LIN {X 0,Y 185.582,Z 221.367,A -85,B 0,C 180,E1 -22200.574,E2 -22200.574} C_VEL
LIN {X 0,Y 185.587,Z 221.368,A -85,B 0,C 180,E1 -22205.381,E2 -22205.381} C_VEL
LIN {X 0,Y 185.674,Z 221.358,A -85,B 0,C 180,E1 -22211.131,E2 -22211.131} C_VEL
LIN {X 0,Y 185.764,Z 221.345,A -85,B 0,C 180,E1 -22216.878,E2 -22216.878} C_VEL
LIN {X 0,Y 186.023,Z 221.31,A -85,B 0,C 180,E1 -22221.307,E2 -22221.307} C_VEL
LIN {X 0,Y 186.206,Z 221.287,A -85,B 0,C 180,E1 -22227.835,E2 -22227.835} C_VEL
LIN {X 0,Y 186.405,Z 221.26,A -85,B 0,C 180,E1 -22229.998,E2 -22229.998} C_VEL
LIN {X 0,Y 185.923,Z 221.325,A -85,B 0,C 180,E1 -22234.334,E2 -22234.334} C_VEL
LIN {X 0,Y 186.006,Z 221.311,A -85,B 0,C 180,E1 -22238.691,E2 -22238.691} C_VEL
LIN {X 0,Y 185.761,Z 221.346,A -85,B 0,C 180,E1 -22243.119,E2 -22243.119} C_VEL
LIN {X 0,Y 185.671,Z 221.357,A -85,B 0,C 180,E1 -22248.866,E2 -22248.866} C_VEL
LIN {X 0,Y 185.596,Z 221.363,A -85,B 0,C 180,E1 -22254.661,E2 -22254.661} C_VEL
LIN {X 0,Y 185.574,Z 221.368,A -85,B 0,C 180,E1 -22259.492,E2 -22259.492} C_VEL
LIN {X 0,Y 185.515,Z 221.375,A -85,B 0,C 180,E1 -22264.626,E2 -22264.626} C_VEL
LIN {X 0,Y 185.562,Z 221.369,A -85,B 0,C 180,E1 -22267.313,E2 -22267.313} C_VEL
LIN {X 0,Y 185.556,Z 221.367,A -85,B 0,C 180,E1 -22270.757,E2 -22270.757} C_VEL
LIN {X 0,Y 185.555,Z 221.371,A -85,B 0,C 180,E1 -22276.022,E2 -22276.022} C_VEL
LIN {X 0,Y 185.527,Z 221.371,A -85,B 0,C 180,E1 -22279.912,E2 -22279.912} C_VEL
LIN {X 0,Y 185.537,Z 221.373,A -85,B 0,C 180,E1 -22282.696,E2 -22282.696} C_VEL
LIN {X 0,Y 185.539,Z 221.371,A -85,B 0,C 180,E1 -22287.975,E2 -22287.975} C_VEL
LIN {X 0,Y 185.575,Z 221.368,A -85,B 0,C 180,E1 -22290.576,E2 -22290.576} C_VEL
LIN {X 0,Y 185.581,Z 221.366,A -85,B 0,C 180,E1 -22295.383,E2 -22295.383} C_VEL
LIN {X 0,Y 185.668,Z 221.356,A -85,B 0,C 180,E1 -22301.133,E2 -22301.133} C_VEL
LIN {X 0,Y 185.688,Z 221.35,A -85,B 0,C 180,E1 -22304.638,E2 -22304.638} C_VEL
LIN {X 0,Y 185.882,Z 221.33,A -85,B 0,C 180,E1 -22309.418,E2 -22309.418} C_VEL
LIN {X 0,Y 185.941,Z 221.32,A -85,B 0,C 180,E1 -22313.49,E2 -22313.49} C_VEL
LIN {X 0,Y 186.2,Z 221.292,A -85,B 0,C 180,E1 -22317.838,E2 -22317.838} C_VEL
LIN {X 0,Y 186.401,Z 221.264,A -85,B 0,C 180,E1 -22320.001,E2 -22320.001} C_VEL
LIN {X 0,Y 185.919,Z 221.324,A -85,B 0,C 180,E1 -22324.337,E2 -22324.337} C_VEL
LIN {X 0,Y 186.009,Z 221.312,A -85,B 0,C 180,E1 -22328.694,E2 -22328.694} C_VEL
LIN {X 0,Y 185.729,Z 221.348,A -85,B 0,C 180,E1 -22333.124,E2 -22333.124} C_VEL
LIN {X 0,Y 185.686,Z 221.352,A -85,B 0,C 180,E1 -22337.626,E2 -22337.626} C_VEL
LIN {X 0,Y 185.593,Z 221.365,A -85,B 0,C 180,E1 -22342.253,E2 -22342.253} C_VEL
LIN {X 0,Y 185.557,Z 221.368,A -85,B 0,C 180,E1 -22347.034,E2 -22347.034} C_VEL
LIN {X 0,Y 185.574,Z 221.37,A -85,B 0,C 180,E1 -22349.495,E2 -22349.495} C_VEL
LIN {X 0,Y 185.495,Z 221.379,A -85,B 0,C 180,E1 -22354.634,E2 -22354.634} C_VEL
LIN {X 0,Y 185.503,Z 221.379,A -85,B 0,C 180,E1 -22357.315,E2 -22357.315} C_VEL
LIN {X 0,Y 185.468,Z 221.383,A -85,B 0,C 180,E1 -22360.726,E2 -22360.726} C_VEL
LIN {X 0,Y 185.457,Z 221.384,A -85,B 0,C 180,E1 -22366.057,E2 -22366.057} C_VEL
LIN {X 0,Y 185.554,Z 221.623,A -85,B 0,C 180,E1 -22368.586,E2 -22368.586} C_VEL
LIN {X 0,Y 188.222,Z 233.304,A -85,B 0,C 180,E1 -22373.317,E2 -22373.317} C_VEL
LIN {X 0,Y 191.21,Z 247.009,A -85,B 0,C 180,E1 -22378.502,E2 -22378.502} C_VEL
LIN {X 0,Y 191.532,Z 248.614,A -85,B 0,C 180,E1 -22379.091,E2 -22379.091} C_VEL
LIN {X 0,Y 190.541,Z 254.381,A -85,B 0,C 180,E1 -22380.972,E2 -22380.972} C_VEL
LIN {X 0,Y 190.999,Z 275.587,A -85,B 0,C 180,E1 -22382.161,E2 -22382.161} C_VEL
LIN {X 0,Y 192.737,Z 304.014,A -85,B 0,C 180,E1 -22383.761,E2 -22383.761} C_VEL
LIN {X 0,Y 191.174,Z 343.448,A -85,B 0,C 180,E1 -22385.757,E2 -22385.757} C_VEL
LIN {X 0,Y 190.275,Z 349.218,A -85,B 0,C 180,E1 -22386.03,E2 -22386.03} C_VEL
LIN {X 0,Y 186.914,Z 358.417,A -85,B 0,C 180,E1 -22386.543,E2 -22386.543} C_VEL
LIN {X 0,Y 183.519,Z 367.45,A -85,B 0,C 180,E1 -22387.317,E2 -22387.317} C_VEL
LIN {X 0,Y 182.429,Z 372.966,A -85,B 0,C 180,E1 -22387.93,E2 -22387.93} C_VEL
LIN {X 0,Y 181.332,Z 384.689,A -85,B 0,C 180,E1 -22389.587,E2 -22389.587} C_VEL
LIN {X 0,Y 180.097,Z 396.698,A -85,B 0,C 180,E1 -22391.811,E2 -22391.811} C_VEL
LIN {X 0,Y 178.971,Z 407.243,A -85,B 0,C 180,E1 -22394.339,E2 -22394.339} C_VEL
LIN {X 0,Y 178.275,Z 415.873,A -85,B 0,C 180,E1 -22396.9,E2 -22396.9} C_VEL
LIN {X 0,Y 177.838,Z 423.688,A -85,B 0,C 180,E1 -22399.758,E2 -22399.758} C_VEL
LIN {X 0,Y 177.753,Z 431.165,A -85,B 0,C 180,E1 -22403.19,E2 -22403.19} C_VEL
LIN {X 0,Y 177.955,Z 436.97,A -85,B 0,C 180,E1 -22406.605,E2 -22406.605} C_VEL
LIN {X 0,Y 178.102,Z 441.236,A -85,B 0,C 180,E1 -22410.002,E2 -22410.002} C_VEL
LIN {X 0,Y 177.77,Z 443.242,A -85,B 0,C 180,E1 -22412.267,E2 -22412.267} C_VEL
LIN {X 0,Y 177.257,Z 444.744,A -85,B 0,C 180,E1 -22414.55,E2 -22414.55} C_VEL
LIN {X 0,Y 176.914,Z 445.823,A -85,B 0,C 180,E1 -22416.846,E2 -22416.846} C_VEL
LIN {X 0,Y 176.939,Z 446.736,A -85,B 0,C 180,E1 -22421.457,E2 -22421.457} C_VEL
LIN {X 0,Y 178.334,Z 446.179,A -85,B 0,C 180,E1 -22426.015,E2 -22426.015} C_VEL
LIN {X 0,Y 181.151,Z 444.075,A -85,B 0,C 180,E1 -22430.438,E2 -22430.438} C_VEL
LIN {X 0,Y 185.157,Z 440.45,A -85,B 0,C 180,E1 -22434.68,E2 -22434.68} C_VEL
LIN {X 0,Y 188.911,Z 436.629,A -85,B 0,C 180,E1 -22437.714,E2 -22437.714} C_VEL
LIN {X 0,Y 193.435,Z 431.743,A -85,B 0,C 180,E1 -22440.576,E2 -22440.576} C_VEL
LIN {X 0,Y 199.599,Z 424.531,A -85,B 0,C 180,E1 -22443.682,E2 -22443.682} C_VEL
LIN {X 0,Y 205.382,Z 416.886,A -85,B 0,C 180,E1 -22446.178,E2 -22446.178} C_VEL
LIN {X 0,Y 211.709,Z 407.374,A -85,B 0,C 180,E1 -22448.495,E2 -22448.495} C_VEL
LIN {X 0,Y 217.437,Z 397.694,A -85,B 0,C 180,E1 -22450.275,E2 -22450.275} C_VEL
LIN {X 0,Y 223.572,Z 385.631,A -85,B 0,C 180,E1 -22451.914,E2 -22451.914} C_VEL
LIN {X 0,Y 227.994,Z 375.107,A -85,B 0,C 180,E1 -22453.002,E2 -22453.002} C_VEL
LIN {X 0,Y 232.578,Z 361.508,A -85,B 0,C 180,E1 -22454.029,E2 -22454.029} C_VEL
LIN {X 0,Y 235.99,Z 347.508,A -85,B 0,C 180,E1 -22454.767,E2 -22454.767} C_VEL
LIN {X 0,Y 240.798,Z 317.9,A -85,B 0,C 180,E1 -22456.017,E2 -22456.017} C_VEL
LIN {X 0,Y 241.066,Z 314.821,A -85,B 0,C 180,E1 -22456.308,E2 -22456.308} C_VEL
LIN {X 0,Y 239.637,Z 310.317,A -85,B 0,C 180,E1 -22458.172,E2 -22458.172} C_VEL
LIN {X 0,Y 238.378,Z 306.264,A -85,B 0,C 180,E1 -22460.344,E2 -22460.344} C_VEL
LIN {X 0,Y 237.037,Z 302.381,A -85,B 0,C 180,E1 -22463.766,E2 -22463.766} C_VEL
LIN {X 0,Y 236.768,Z 301.25,A -85,B 0,C 180,E1 -22465.668,E2 -22465.668} C_VEL
LIN {X 0,Y 236.704,Z 300.974,A -85,B 0,C 180,E1 -22467.693,E2 -22467.693} C_VEL
LIN {X 0,Y 237.19,Z 301.52,A -85,B 0,C 180,E1 -22470.349,E2 -22470.349} C_VEL
LIN {X 0,Y 238.419,Z 303.667,A -85,B 0,C 180,E1 -22473.28,E2 -22473.28} C_VEL
LIN {X 0,Y 240.206,Z 307.592,A -85,B 0,C 180,E1 -22476.073,E2 -22476.073} C_VEL
LIN {X 0,Y 241.314,Z 310.279,A -85,B 0,C 180,E1 -22477.425,E2 -22477.425} C_VEL
LIN {X 0,Y 236.461,Z 338.426,A -85,B 0,C 180,E1 -22478.792,E2 -22478.792} C_VEL
LIN {X 0,Y 233.294,Z 351.201,A -85,B 0,C 180,E1 -22479.73,E2 -22479.73} C_VEL
LIN {X 0,Y 229.171,Z 363.637,A -85,B 0,C 180,E1 -22480.983,E2 -22480.983} C_VEL
LIN {X 0,Y 224.538,Z 374.681,A -85,B 0,C 180,E1 -22482.466,E2 -22482.466} C_VEL
LIN {X 0,Y 219.655,Z 384.181,A -85,B 0,C 180,E1 -22484.128,E2 -22484.128} C_VEL
LIN {X 0,Y 214.005,Z 393.392,A -85,B 0,C 180,E1 -22486.225,E2 -22486.225} C_VEL
LIN {X 0,Y 208.873,Z 400.55,A -85,B 0,C 180,E1 -22488.352,E2 -22488.352} C_VEL
LIN {X 0,Y 203.977,Z 406.361,A -85,B 0,C 180,E1 -22490.58,E2 -22490.58} C_VEL
LIN {X 0,Y 199.59,Z 410.86,A -85,B 0,C 180,E1 -22492.879,E2 -22492.879} C_VEL
LIN {X 0,Y 194.612,Z 415.134,A -85,B 0,C 180,E1 -22495.857,E2 -22495.857} C_VEL
LIN {X 0,Y 189.772,Z 418.269,A -85,B 0,C 180,E1 -22499.324,E2 -22499.324} C_VEL
LIN {X 0,Y 186.483,Z 419.638,A -85,B 0,C 180,E1 -22502.159,E2 -22502.159} C_VEL
LIN {X 0,Y 183.501,Z 420.12,A -85,B 0,C 180,E1 -22505.252,E2 -22505.252} C_VEL
LIN {X 0,Y 180.779,Z 419.378,A -85,B 0,C 180,E1 -22508.945,E2 -22508.945} C_VEL
LIN {X 0,Y 179.319,Z 418.115,A -85,B 0,C 180,E1 -22511.525,E2 -22511.525} C_VEL
LIN {X 0,Y 177.929,Z 415.513,A -85,B 0,C 180,E1 -22514.876,E2 -22514.876} C_VEL
LIN {X 0,Y 177.063,Z 411.424,A -85,B 0,C 180,E1 -22518.513,E2 -22518.513} C_VEL
LIN {X 0,Y 176.816,Z 405.855,A -85,B 0,C 180,E1 -22522.184,E2 -22522.184} C_VEL
LIN {X 0,Y 177.175,Z 398.545,A -85,B 0,C 180,E1 -22525.869,E2 -22525.869} C_VEL
LIN {X 0,Y 177.738,Z 390.602,A -85,B 0,C 180,E1 -22528.993,E2 -22528.993} C_VEL
LIN {X 0,Y 178.494,Z 381.753,A -85,B 0,C 180,E1 -22531.776,E2 -22531.776} C_VEL
LIN {X 0,Y 179.446,Z 371.889,A -85,B 0,C 180,E1 -22534.26,E2 -22534.26} C_VEL
LIN {X 0,Y 180.458,Z 361.055,A -85,B 0,C 180,E1 -22536.434,E2 -22536.434} C_VEL
LIN {X 0,Y 181.491,Z 349.211,A -85,B 0,C 180,E1 -22538.284,E2 -22538.284} C_VEL
LIN {X 0,Y 182.352,Z 337.137,A -85,B 0,C 180,E1 -22539.692,E2 -22539.692} C_VEL
LIN {X 0,Y 182.996,Z 323.953,A -85,B 0,C 180,E1 -22540.758,E2 -22540.758} C_VEL
LIN {X 0,Y 185.457,Z 265.599,A -85,B 0,C 180,E1 -22544.188,E2 -22544.188} C_VEL
LIN {X 0,Y 182.652,Z 241.648,A -85,B 0,C 180,E1 -22545.793,E2 -22545.793} C_VEL
LIN {X 0,Y 181.654,Z 237.511,A -85,B 0,C 180,E1 -22546.212,E2 -22546.212} C_VEL
LIN {X 0,Y 179.188,Z 225.225,A -85,B 0,C 180,E1 -22551.666,E2 -22551.666} C_VEL
LIN {X 0,Y 178.573,Z 222.387,A -85,B 0,C 180,E1 -22553.103,E2 -22553.103} C_VEL
LIN {X 0,Y 178.489,Z 222.252,A -85,B 0,C 180,E1 -22556.546,E2 -22556.546} C_VEL
LIN {X 0,Y 178.523,Z 222.248,A -85,B 0,C 180,E1 -22560.005,E2 -22560.005} C_VEL
LIN {X 0,Y 178.534,Z 222.244,A -85,B 0,C 180,E1 -22564.874,E2 -22564.874} C_VEL
LIN {X 0,Y 178.622,Z 222.235,A -85,B 0,C 180,E1 -22570.782,E2 -22570.782} C_VEL
LIN {X 0,Y 178.68,Z 222.226,A -85,B 0,C 180,E1 -22576.348,E2 -22576.348} C_VEL
LIN {X 0,Y 178.973,Z 222.188,A -85,B 0,C 180,E1 -22580.961,E2 -22580.961} C_VEL
LIN {X 0,Y 179.152,Z 222.166,A -85,B 0,C 180,E1 -22587.75,E2 -22587.75} C_VEL
LIN {X 0,Y 179.368,Z 222.137,A -85,B 0,C 180,E1 -22589.998,E2 -22589.998} C_VEL
LIN {X 0,Y 178.871,Z 222.204,A -85,B 0,C 180,E1 -22594.505,E2 -22594.505} C_VEL
LIN {X 0,Y 178.956,Z 222.191,A -85,B 0,C 180,E1 -22599.036,E2 -22599.036} C_VEL
LIN {X 0,Y 178.678,Z 222.226,A -85,B 0,C 180,E1 -22603.649,E2 -22603.649} C_VEL
LIN {X 0,Y 178.619,Z 222.235,A -85,B 0,C 180,E1 -22609.215,E2 -22609.215} C_VEL
LIN {X 0,Y 178.53,Z 222.243,A -85,B 0,C 180,E1 -22615.123,E2 -22615.123} C_VEL
LIN {X 0,Y 178.474,Z 222.252,A -85,B 0,C 180,E1 -22620.789,E2 -22620.789} C_VEL
LIN {X 0,Y 178.479,Z 222.248,A -85,B 0,C 180,E1 -22624.219,E2 -22624.219} C_VEL
LIN {X 0,Y 178.467,Z 222.252,A -85,B 0,C 180,E1 -22629.053,E2 -22629.053} C_VEL
LIN {X 0,Y 178.494,Z 222.246,A -85,B 0,C 180,E1 -22632.015,E2 -22632.015} C_VEL
LIN {X 0,Y 178.51,Z 222.248,A -85,B 0,C 180,E1 -22635.124,E2 -22635.124} C_VEL
LIN {X 0,Y 178.478,Z 222.251,A -85,B 0,C 180,E1 -22638.429,E2 -22638.429} C_VEL
LIN {X 0,Y 178.444,Z 222.257,A -85,B 0,C 180,E1 -22643.789,E2 -22643.789} C_VEL
LIN {X 0,Y 178.485,Z 222.25,A -85,B 0,C 180,E1 -22646.548,E2 -22646.548} C_VEL
LIN {X 0,Y 178.516,Z 222.246,A -85,B 0,C 180,E1 -22650.006,E2 -22650.006} C_VEL
LIN {X 0,Y 178.528,Z 222.244,A -85,B 0,C 180,E1 -22654.876,E2 -22654.876} C_VEL
LIN {X 0,Y 178.617,Z 222.234,A -85,B 0,C 180,E1 -22660.784,E2 -22660.784} C_VEL
LIN {X 0,Y 178.651,Z 222.229,A -85,B 0,C 180,E1 -22666.348,E2 -22666.348} C_VEL
LIN {X 0,Y 178.905,Z 222.198,A -85,B 0,C 180,E1 -22670.961,E2 -22670.961} C_VEL
LIN {X 0,Y 179.146,Z 222.171,A -85,B 0,C 180,E1 -22677.753,E2 -22677.753} C_VEL
LIN {X 0,Y 179.364,Z 222.141,A -85,B 0,C 180,E1 -22680.001,E2 -22680.001} C_VEL
LIN {X 0,Y 178.868,Z 222.202,A -85,B 0,C 180,E1 -22684.508,E2 -22684.508} C_VEL
LIN {X 0,Y 178.958,Z 222.191,A -85,B 0,C 180,E1 -22689.039,E2 -22689.039} C_VEL
LIN {X 0,Y 178.656,Z 222.232,A -85,B 0,C 180,E1 -22693.653,E2 -22693.653} C_VEL
LIN {X 0,Y 178.619,Z 222.231,A -85,B 0,C 180,E1 -22699.218,E2 -22699.218} C_VEL
LIN {X 0,Y 178.531,Z 222.247,A -85,B 0,C 180,E1 -22705.126,E2 -22705.126} C_VEL
LIN {X 0,Y 178.474,Z 222.254,A -85,B 0,C 180,E1 -22710.793,E2 -22710.793} C_VEL
LIN {X 0,Y 178.481,Z 222.252,A -85,B 0,C 180,E1 -22714.221,E2 -22714.221} C_VEL
LIN {X 0,Y 178.392,Z 222.264,A -85,B 0,C 180,E1 -22719.077,E2 -22719.077} C_VEL
LIN {X 0,Y 178.395,Z 222.263,A -85,B 0,C 180,E1 -22722.047,E2 -22722.047} C_VEL
LIN {X 0,Y 178.391,Z 222.265,A -85,B 0,C 180,E1 -22725.166,E2 -22725.166} C_VEL
LIN {X 0,Y 178.502,Z 222.537,A -85,B 0,C 180,E1 -22728.094,E2 -22728.094} C_VEL
LIN {X 0,Y 181.016,Z 233.563,A -85,B 0,C 180,E1 -22732.742,E2 -22732.742} C_VEL
LIN {X 0,Y 184.108,Z 247.761,A -85,B 0,C 180,E1 -22738.342,E2 -22738.342} C_VEL
LIN {X 0,Y 184.459,Z 249.623,A -85,B 0,C 180,E1 -22739.048,E2 -22739.048} C_VEL
LIN {X 0,Y 183.628,Z 253.91,A -85,B 0,C 180,E1 -22740.496,E2 -22740.496} C_VEL
LIN {X 0,Y 183.824,Z 271.879,A -85,B 0,C 180,E1 -22741.565,E2 -22741.565} C_VEL
LIN {X 0,Y 185.717,Z 304.253,A -85,B 0,C 180,E1 -22743.45,E2 -22743.45} C_VEL
LIN {X 0,Y 183.695,Z 355.631,A -85,B 0,C 180,E1 -22746.271,E2 -22746.271} C_VEL
LIN {X 0,Y 182.99,Z 367.173,A -85,B 0,C 180,E1 -22747.282,E2 -22747.282} C_VEL
LIN {X 0,Y 182.429,Z 372.966,A -85,B 0,C 180,E1 -22747.93,E2 -22747.93} C_VEL
LIN {X 0,Y 181.253,Z 378.336,A -85,B 0,C 180,E1 -22748.614,E2 -22748.614} C_VEL
LIN {X 0,Y 177.603,Z 386.618,A -85,B 0,C 180,E1 -22749.908,E2 -22749.908} C_VEL
LIN {X 0,Y 173.919,Z 394.533,A -85,B 0,C 180,E1 -22751.478,E2 -22751.478} C_VEL
LIN {X 0,Y 172.705,Z 399.312,A -85,B 0,C 180,E1 -22752.57,E2 -22752.57} C_VEL
LIN {X 0,Y 171.627,Z 409.102,A -85,B 0,C 180,E1 -22755.173,E2 -22755.173} C_VEL
LIN {X 0,Y 171.042,Z 418.092,A -85,B 0,C 180,E1 -22758.146,E2 -22758.146} C_VEL
LIN {X 0,Y 170.693,Z 425.475,A -85,B 0,C 180,E1 -22761.182,E2 -22761.182} C_VEL
LIN {X 0,Y 170.828,Z 432.261,A -85,B 0,C 180,E1 -22764.69,E2 -22764.69} C_VEL
LIN {X 0,Y 171.081,Z 436.784,A -85,B 0,C 180,E1 -22767.647,E2 -22767.647} C_VEL
LIN {X 0,Y 171.163,Z 439.627,A -85,B 0,C 180,E1 -22770.002,E2 -22770.002} C_VEL
LIN {X 0,Y 170.795,Z 441.824,A -85,B 0,C 180,E1 -22772.36,E2 -22772.36} C_VEL
LIN {X 0,Y 169.927,Z 444.564,A -85,B 0,C 180,E1 -22776.959,E2 -22776.959} C_VEL
LIN {X 0,Y 169.771,Z 445.424,A -85,B 0,C 180,E1 -22779.533,E2 -22779.533} C_VEL
LIN {X 0,Y 170.562,Z 445.861,A -85,B 0,C 180,E1 -22784.315,E2 -22784.315} C_VEL
LIN {X 0,Y 172.832,Z 444.823,A -85,B 0,C 180,E1 -22788.986,E2 -22788.986} C_VEL
LIN {X 0,Y 174.502,Z 443.763,A -85,B 0,C 180,E1 -22791.254,E2 -22791.254} C_VEL
LIN {X 0,Y 178.698,Z 440.432,A -85,B 0,C 180,E1 -22795.635,E2 -22795.635} C_VEL
LIN {X 0,Y 182.654,Z 436.866,A -85,B 0,C 180,E1 -22798.75,E2 -22798.75} C_VEL
LIN {X 0,Y 187.39,Z 432.327,A -85,B 0,C 180,E1 -22801.674,E2 -22801.674} C_VEL
LIN {X 0,Y 193.804,Z 425.594,A -85,B 0,C 180,E1 -22804.832,E2 -22804.832} C_VEL
LIN {X 0,Y 199.795,Z 418.312,A -85,B 0,C 180,E1 -22807.359,E2 -22807.359} C_VEL
LIN {X 0,Y 206.341,Z 409.483,A -85,B 0,C 180,E1 -22809.691,E2 -22809.691} C_VEL
LIN {X 0,Y 212.824,Z 399.443,A -85,B 0,C 180,E1 -22811.651,E2 -22811.651} C_VEL
LIN {X 0,Y 219.127,Z 388.06,A -85,B 0,C 180,E1 -22813.28,E2 -22813.28} C_VEL
LIN {X 0,Y 225.032,Z 375.094,A -85,B 0,C 180,E1 -22814.645,E2 -22814.645} C_VEL
LIN {X 0,Y 229.762,Z 361.936,A -85,B 0,C 180,E1 -22815.644,E2 -22815.644} C_VEL
LIN {X 0,Y 233.3,Z 348.771,A -85,B 0,C 180,E1 -22816.349,E2 -22816.349} C_VEL
LIN {X 0,Y 238.354,Z 319.482,A -85,B 0,C 180,E1 -22817.571,E2 -22817.571} C_VEL
LIN {X 0,Y 237.48,Z 316.125,A -85,B 0,C 180,E1 -22819.03,E2 -22819.03} C_VEL
LIN {X 0,Y 236.531,Z 312.836,A -85,B 0,C 180,E1 -22820.823,E2 -22820.823} C_VEL
LIN {X 0,Y 235.44,Z 309.191,A -85,B 0,C 180,E1 -22824.071,E2 -22824.071} C_VEL
LIN {X 0,Y 235.228,Z 308.105,A -85,B 0,C 180,E1 -22826,E2 -22826} C_VEL
LIN {X 0,Y 235.265,Z 307.946,A -85,B 0,C 180,E1 -22828.29,E2 -22828.29} C_VEL
LIN {X 0,Y 235.798,Z 308.729,A -85,B 0,C 180,E1 -22830.768,E2 -22830.768} C_VEL
LIN {X 0,Y 236.725,Z 310.562,A -85,B 0,C 180,E1 -22833.071,E2 -22833.071} C_VEL
LIN {X 0,Y 238.329,Z 314.413,A -85,B 0,C 180,E1 -22835.762,E2 -22835.762} C_VEL
LIN {X 0,Y 238.469,Z 314.81,A -85,B 0,C 180,E1 -22835.983,E2 -22835.983} C_VEL
LIN {X 0,Y 233.809,Z 340.377,A -85,B 0,C 180,E1 -22837.239,E2 -22837.239} C_VEL
LIN {X 0,Y 230.54,Z 352.77,A -85,B 0,C 180,E1 -22838.168,E2 -22838.168} C_VEL
LIN {X 0,Y 226.548,Z 364.138,A -85,B 0,C 180,E1 -22839.296,E2 -22839.296} C_VEL
LIN {X 0,Y 221.7,Z 375.004,A -85,B 0,C 180,E1 -22840.725,E2 -22840.725} C_VEL
LIN {X 0,Y 216.176,Z 385.248,A -85,B 0,C 180,E1 -22842.498,E2 -22842.498} C_VEL
LIN {X 0,Y 210.426,Z 394.163,A -85,B 0,C 180,E1 -22844.502,E2 -22844.502} C_VEL
LIN {X 0,Y 203.934,Z 402.509,A -85,B 0,C 180,E1 -22847.055,E2 -22847.055} C_VEL
LIN {X 0,Y 197.772,Z 409.059,A -85,B 0,C 180,E1 -22849.764,E2 -22849.764} C_VEL
LIN {X 0,Y 192.551,Z 413.748,A -85,B 0,C 180,E1 -22852.502,E2 -22852.502} C_VEL
LIN {X 0,Y 187.239,Z 417.47,A -85,B 0,C 180,E1 -22855.694,E2 -22855.694} C_VEL
LIN {X 0,Y 182.762,Z 419.768,A -85,B 0,C 180,E1 -22858.94,E2 -22858.94} C_VEL
LIN {X 0,Y 179.014,Z 420.831,A -85,B 0,C 180,E1 -22862.249,E2 -22862.249} C_VEL
LIN {X 0,Y 176.384,Z 420.838,A -85,B 0,C 180,E1 -22865.037,E2 -22865.037} C_VEL
LIN {X 0,Y 174.945,Z 420.446,A -85,B 0,C 180,E1 -22866.921,E2 -22866.921} C_VEL
LIN {X 0,Y 173.334,Z 419.463,A -85,B 0,C 180,E1 -22869.333,E2 -22869.333} C_VEL
LIN {X 0,Y 171.474,Z 416.992,A -85,B 0,C 180,E1 -22873.026,E2 -22873.026} C_VEL
LIN {X 0,Y 170.263,Z 413.258,A -85,B 0,C 180,E1 -22876.793,E2 -22876.793} C_VEL
LIN {X 0,Y 169.78,Z 408.067,A -85,B 0,C 180,E1 -22880.6,E2 -22880.6} C_VEL
LIN {X 0,Y 169.845,Z 402.477,A -85,B 0,C 180,E1 -22883.792,E2 -22883.792} C_VEL
LIN {X 0,Y 170.308,Z 395.497,A -85,B 0,C 180,E1 -22886.995,E2 -22886.995} C_VEL
LIN {X 0,Y 170.985,Z 386.404,A -85,B 0,C 180,E1 -22890.324,E2 -22890.324} C_VEL
LIN {X 0,Y 172.022,Z 375.426,A -85,B 0,C 180,E1 -22893.472,E2 -22893.472} C_VEL
LIN {X 0,Y 173.162,Z 363.57,A -85,B 0,C 180,E1 -22896.1,E2 -22896.1} C_VEL
LIN {X 0,Y 174.224,Z 351.436,A -85,B 0,C 180,E1 -22898.146,E2 -22898.146} C_VEL
LIN {X 0,Y 175.175,Z 338.681,A -85,B 0,C 180,E1 -22899.746,E2 -22899.746} C_VEL
LIN {X 0,Y 175.85,Z 326.101,A -85,B 0,C 180,E1 -22900.854,E2 -22900.854} C_VEL
LIN {X 0,Y 178.443,Z 266.016,A -85,B 0,C 180,E1 -22904.55,E2 -22904.55} C_VEL
LIN {X 0,Y 175.792,Z 243.119,A -85,B 0,C 180,E1 -22906.165,E2 -22906.165} C_VEL
LIN {X 0,Y 174.512,Z 237.87,A -85,B 0,C 180,E1 -22906.67,E2 -22906.67} C_VEL
LIN {X 0,Y 172.038,Z 225.846,A -85,B 0,C 180,E1 -22912.208,E2 -22912.208} C_VEL
LIN {X 0,Y 171.539,Z 223.201,A -85,B 0,C 180,E1 -22913.643,E2 -22913.643} C_VEL
LIN {X 0,Y 171.458,Z 223.129,A -85,B 0,C 180,E1 -22919.402,E2 -22919.402} C_VEL
LIN {X 0,Y 171.469,Z 223.124,A -85,B 0,C 180,E1 -22924.382,E2 -22924.382} C_VEL
LIN {X 0,Y 171.578,Z 223.112,A -85,B 0,C 180,E1 -22930.87,E2 -22930.87} C_VEL
LIN {X 0,Y 171.593,Z 223.11,A -85,B 0,C 180,E1 -22935.773,E2 -22935.773} C_VEL
LIN {X 0,Y 171.906,Z 223.068,A -85,B 0,C 180,E1 -22940.587,E2 -22940.587} C_VEL
LIN {X 0,Y 171.823,Z 223.083,A -85,B 0,C 180,E1 -22945.306,E2 -22945.306} C_VEL
LIN {X 0,Y 172.331,Z 223.013,A -85,B 0,C 180,E1 -22949.998,E2 -22949.998} C_VEL
LIN {X 0,Y 171.82,Z 223.083,A -85,B 0,C 180,E1 -22954.691,E2 -22954.691} C_VEL
LIN {X 0,Y 171.885,Z 223.072,A -85,B 0,C 180,E1 -22959.411,E2 -22959.411} C_VEL
LIN {X 0,Y 171.591,Z 223.109,A -85,B 0,C 180,E1 -22964.224,E2 -22964.224} C_VEL
LIN {X 0,Y 171.54,Z 223.116,A -85,B 0,C 180,E1 -22969.561,E2 -22969.561} C_VEL
LIN {X 0,Y 171.464,Z 223.122,A -85,B 0,C 180,E1 -22975.615,E2 -22975.615} C_VEL
LIN {X 0,Y 171.437,Z 223.13,A -85,B 0,C 180,E1 -22980.586,E2 -22980.586} C_VEL
LIN {X 0,Y 171.399,Z 223.133,A -85,B 0,C 180,E1 -22985.031,E2 -22985.031} C_VEL
LIN {X 0,Y 171.421,Z 223.131,A -85,B 0,C 180,E1 -22988.836,E2 -22988.836} C_VEL
LIN {X 0,Y 171.436,Z 223.129,A -85,B 0,C 180,E1 -22994.177,E2 -22994.177} C_VEL
LIN {X 0,Y 171.395,Z 223.131,A -85,B 0,C 180,E1 -22999,E2 -22999} C_VEL
LIN {X 0,Y 171.415,Z 223.131,A -85,B 0,C 180,E1 -23002.05,E2 -23002.05} C_VEL
LIN {X 0,Y 171.405,Z 223.133,A -85,B 0,C 180,E1 -23005.086,E2 -23005.086} C_VEL
LIN {X 0,Y 171.443,Z 223.128,A -85,B 0,C 180,E1 -23010.535,E2 -23010.535} C_VEL
LIN {X 0,Y 171.451,Z 223.126,A -85,B 0,C 180,E1 -23015.802,E2 -23015.802} C_VEL
LIN {X 0,Y 171.573,Z 223.112,A -85,B 0,C 180,E1 -23020.872,E2 -23020.872} C_VEL
LIN {X 0,Y 171.569,Z 223.109,A -85,B 0,C 180,E1 -23025.773,E2 -23025.773} C_VEL
LIN {X 0,Y 171.842,Z 223.078,A -85,B 0,C 180,E1 -23030.586,E2 -23030.586} C_VEL
LIN {X 0,Y 171.809,Z 223.08,A -85,B 0,C 180,E1 -23035.308,E2 -23035.308} C_VEL
LIN {X 0,Y 172.327,Z 223.017,A -85,B 0,C 180,E1 -23040.001,E2 -23040.001} C_VEL
LIN {X 0,Y 171.817,Z 223.081,A -85,B 0,C 180,E1 -23044.694,E2 -23044.694} C_VEL
LIN {X 0,Y 171.886,Z 223.071,A -85,B 0,C 180,E1 -23049.414,E2 -23049.414} C_VEL
LIN {X 0,Y 171.573,Z 223.112,A -85,B 0,C 180,E1 -23054.229,E2 -23054.229} C_VEL
LIN {X 0,Y 171.54,Z 223.114,A -85,B 0,C 180,E1 -23059.564,E2 -23059.564} C_VEL
LIN {X 0,Y 171.465,Z 223.124,A -85,B 0,C 180,E1 -23065.618,E2 -23065.618} C_VEL
LIN {X 0,Y 171.436,Z 223.13,A -85,B 0,C 180,E1 -23070.587,E2 -23070.587} C_VEL
LIN {X 0,Y 171.39,Z 223.138,A -85,B 0,C 180,E1 -23075.037,E2 -23075.037} C_VEL
LIN {X 0,Y 171.355,Z 223.14,A -85,B 0,C 180,E1 -23078.809,E2 -23078.809} C_VEL
LIN {X 0,Y 171.318,Z 223.145,A -85,B 0,C 180,E1 -23084.22,E2 -23084.22} C_VEL
LIN {X 0,Y 171.43,Z 223.387,A -85,B 0,C 180,E1 -23087.557,E2 -23087.557} C_VEL
LIN {X 0,Y 173.923,Z 234.398,A -85,B 0,C 180,E1 -23092.392,E2 -23092.392} C_VEL
LIN {X 0,Y 176.673,Z 246.948,A -85,B 0,C 180,E1 -23097.546,E2 -23097.546} C_VEL
LIN {X 0,Y 177.32,Z 250.582,A -85,B 0,C 180,E1 -23098.988,E2 -23098.988} C_VEL
LIN {X 0,Y 176.665,Z 253.766,A -85,B 0,C 180,E1 -23100.076,E2 -23100.076} C_VEL
LIN {X 0,Y 176.965,Z 275.277,A -85,B 0,C 180,E1 -23101.375,E2 -23101.375} C_VEL
LIN {X 0,Y 178.66,Z 304.843,A -85,B 0,C 180,E1 -23103.185,E2 -23103.185} C_VEL
LIN {X 0,Y 176.634,Z 355.237,A -85,B 0,C 180,E1 -23106.081,E2 -23106.081} C_VEL
LIN {X 0,Y 175.853,Z 367.669,A -85,B 0,C 180,E1 -23107.234,E2 -23107.234} C_VEL
LIN {X 0,Y 174.764,Z 379.495,A -85,B 0,C 180,E1 -23108.783,E2 -23108.783} C_VEL
LIN {X 0,Y 173.565,Z 391.128,A -85,B 0,C 180,E1 -23110.794,E2 -23110.794} C_VEL
LIN {X 0,Y 172.705,Z 399.312,A -85,B 0,C 180,E1 -23112.57,E2 -23112.57} C_VEL
LIN {X 0,Y 171.497,Z 403.924,A -85,B 0,C 180,E1 -23113.744,E2 -23113.744} C_VEL
LIN {X 0,Y 167.932,Z 410.724,A -85,B 0,C 180,E1 -23115.871,E2 -23115.871} C_VEL
LIN {X 0,Y 164.649,Z 417.032,A -85,B 0,C 180,E1 -23118.28,E2 -23118.28} C_VEL
LIN {X 0,Y 163.89,Z 420.781,A -85,B 0,C 180,E1 -23119.851,E2 -23119.851} C_VEL
LIN {X 0,Y 163.813,Z 427.926,A -85,B 0,C 180,E1 -23123.226,E2 -23123.226} C_VEL
LIN {X 0,Y 163.994,Z 433.162,A -85,B 0,C 180,E1 -23126.316,E2 -23126.316} C_VEL
LIN {X 0,Y 164.224,Z 436.539,A -85,B 0,C 180,E1 -23128.776,E2 -23128.776} C_VEL
LIN {X 0,Y 164.07,Z 439.23,A -85,B 0,C 180,E1 -23131.229,E2 -23131.229} C_VEL
LIN {X 0,Y 163.265,Z 442.071,A -85,B 0,C 180,E1 -23134.941,E2 -23134.941} C_VEL
LIN {X 0,Y 162.898,Z 443.394,A -85,B 0,C 180,E1 -23137.438,E2 -23137.438} C_VEL
LIN {X 0,Y 163.031,Z 444.836,A -85,B 0,C 180,E1 -23142.449,E2 -23142.449} C_VEL
LIN {X 0,Y 164.701,Z 444.853,A -85,B 0,C 180,E1 -23147.381,E2 -23147.381} C_VEL
LIN {X 0,Y 167.872,Z 443.361,A -85,B 0,C 180,E1 -23152.136,E2 -23152.136} C_VEL
LIN {X 0,Y 172.304,Z 440.396,A -85,B 0,C 180,E1 -23156.66,E2 -23156.66} C_VEL
LIN {X 0,Y 176.472,Z 437.138,A -85,B 0,C 180,E1 -23159.857,E2 -23159.857} C_VEL
LIN {X 0,Y 181.421,Z 432.9,A -85,B 0,C 180,E1 -23162.845,E2 -23162.845} C_VEL
LIN {X 0,Y 188.073,Z 426.539,A -85,B 0,C 180,E1 -23166.056,E2 -23166.056} C_VEL
LIN {X 0,Y 195.386,Z 418.545,A -85,B 0,C 180,E1 -23169.012,E2 -23169.012} C_VEL
LIN {X 0,Y 202.217,Z 409.905,A -85,B 0,C 180,E1 -23171.327,E2 -23171.327} C_VEL
LIN {X 0,Y 208.325,Z 401.157,A -85,B 0,C 180,E1 -23173.091,E2 -23173.091} C_VEL
LIN {X 0,Y 214.867,Z 390.474,A -85,B 0,C 180,E1 -23174.688,E2 -23174.688} C_VEL
LIN {X 0,Y 220.892,Z 378.54,A -85,B 0,C 180,E1 -23176.043,E2 -23176.043} C_VEL
LIN {X 0,Y 225.779,Z 366.558,A -85,B 0,C 180,E1 -23177.014,E2 -23177.014} C_VEL
LIN {X 0,Y 229.494,Z 354.984,A -85,B 0,C 180,E1 -23177.726,E2 -23177.726} C_VEL
LIN {X 0,Y 232.917,Z 340.14,A -85,B 0,C 180,E1 -23178.4,E2 -23178.4} C_VEL
LIN {X 0,Y 235.831,Z 323.61,A -85,B 0,C 180,E1 -23179.051,E2 -23179.051} C_VEL
LIN {X 0,Y 234.755,Z 319.39,A -85,B 0,C 180,E1 -23181.322,E2 -23181.322} C_VEL
LIN {X 0,Y 233.865,Z 315.922,A -85,B 0,C 180,E1 -23184.463,E2 -23184.463} C_VEL
LIN {X 0,Y 233.706,Z 315.024,A -85,B 0,C 180,E1 -23186.107,E2 -23186.107} C_VEL
LIN {X 0,Y 233.9,Z 315.046,A -85,B 0,C 180,E1 -23189.282,E2 -23189.282} C_VEL
LIN {X 0,Y 234.601,Z 316.36,A -85,B 0,C 180,E1 -23191.709,E2 -23191.709} C_VEL
LIN {X 0,Y 235.172,Z 317.943,A -85,B 0,C 180,E1 -23193.21,E2 -23193.21} C_VEL
LIN {X 0,Y 235.917,Z 319.667,A -85,B 0,C 180,E1 -23194.519,E2 -23194.519} C_VEL
LIN {X 0,Y 231.768,Z 341.207,A -85,B 0,C 180,E1 -23195.583,E2 -23195.583} C_VEL
LIN {X 0,Y 228.525,Z 352.861,A -85,B 0,C 180,E1 -23196.433,E2 -23196.433} C_VEL
LIN {X 0,Y 223.945,Z 365.222,A -85,B 0,C 180,E1 -23197.633,E2 -23197.633} C_VEL
LIN {X 0,Y 218.891,Z 376.078,A -85,B 0,C 180,E1 -23199.032,E2 -23199.032} C_VEL
LIN {X 0,Y 213.175,Z 386.092,A -85,B 0,C 180,E1 -23200.75,E2 -23200.75} C_VEL
LIN {X 0,Y 206.786,Z 395.306,A -85,B 0,C 180,E1 -23202.824,E2 -23202.824} C_VEL
LIN {X 0,Y 200.216,Z 403.332,A -85,B 0,C 180,E1 -23205.256,E2 -23205.256} C_VEL
LIN {X 0,Y 194.201,Z 409.37,A -85,B 0,C 180,E1 -23207.721,E2 -23207.721} C_VEL
LIN {X 0,Y 188.725,Z 413.993,A -85,B 0,C 180,E1 -23210.352,E2 -23210.352} C_VEL
LIN {X 0,Y 182.89,Z 417.964,A -85,B 0,C 180,E1 -23213.603,E2 -23213.603} C_VEL
LIN {X 0,Y 179.865,Z 419.563,A -85,B 0,C 180,E1 -23215.517,E2 -23215.517} C_VEL
LIN {X 0,Y 175.762,Z 421.116,A -85,B 0,C 180,E1 -23218.51,E2 -23218.51} C_VEL
LIN {X 0,Y 171.494,Z 421.763,A -85,B 0,C 180,E1 -23222.348,E2 -23222.348} C_VEL
LIN {X 0,Y 169.266,Z 421.437,A -85,B 0,C 180,E1 -23224.79,E2 -23224.79} C_VEL
LIN {X 0,Y 167.454,Z 420.637,A -85,B 0,C 180,E1 -23227.232,E2 -23227.232} C_VEL
LIN {X 0,Y 164.968,Z 418.05,A -85,B 0,C 180,E1 -23231.516,E2 -23231.516} C_VEL
LIN {X 0,Y 163.644,Z 414.938,A -85,B 0,C 180,E1 -23234.931,E2 -23234.931} C_VEL
LIN {X 0,Y 162.824,Z 409.74,A -85,B 0,C 180,E1 -23239.149,E2 -23239.149} C_VEL
LIN {X 0,Y 162.741,Z 402.728,A -85,B 0,C 180,E1 -23243.412,E2 -23243.412} C_VEL
LIN {X 0,Y 163.211,Z 395.336,A -85,B 0,C 180,E1 -23246.88,E2 -23246.88} C_VEL
LIN {X 0,Y 163.89,Z 386.307,A -85,B 0,C 180,E1 -23250.255,E2 -23250.255} C_VEL
LIN {X 0,Y 164.822,Z 376.188,A -85,B 0,C 180,E1 -23253.26,E2 -23253.26} C_VEL
LIN {X 0,Y 165.955,Z 364.47,A -85,B 0,C 180,E1 -23255.985,E2 -23255.985} C_VEL
LIN {X 0,Y 167.126,Z 351.664,A -85,B 0,C 180,E1 -23258.259,E2 -23258.259} C_VEL
LIN {X 0,Y 168.13,Z 338.345,A -85,B 0,C 180,E1 -23259.991,E2 -23259.991} C_VEL
LIN {X 0,Y 168.844,Z 325.1,A -85,B 0,C 180,E1 -23261.171,E2 -23261.171} C_VEL
LIN {X 0,Y 171.463,Z 266.646,A -85,B 0,C 180,E1 -23264.92,E2 -23264.92} C_VEL
LIN {X 0,Y 168.88,Z 244.508,A -85,B 0,C 180,E1 -23266.53,E2 -23266.53} C_VEL
LIN {X 0,Y 167.382,Z 238.271,A -85,B 0,C 180,E1 -23267.129,E2 -23267.129} C_VEL
LIN {X 0,Y 164.992,Z 226.774,A -85,B 0,C 180,E1 -23272.626,E2 -23272.626} C_VEL
LIN {X 0,Y 164.475,Z 224.096,A -85,B 0,C 180,E1 -23274.124,E2 -23274.124} C_VEL
LIN {X 0,Y 164.406,Z 224.007,A -85,B 0,C 180,E1 -23279.136,E2 -23279.136} C_VEL
LIN {X 0,Y 164.416,Z 224.002,A -85,B 0,C 180,E1 -23284.692,E2 -23284.692} C_VEL
LIN {X 0,Y 164.484,Z 223.996,A -85,B 0,C 180,E1 -23290.049,E2 -23290.049} C_VEL
LIN {X 0,Y 164.535,Z 223.988,A -85,B 0,C 180,E1 -23295.149,E2 -23295.149} C_VEL
LIN {X 0,Y 164.849,Z 223.946,A -85,B 0,C 180,E1 -23300.18,E2 -23300.18} C_VEL
LIN {X 0,Y 164.773,Z 223.961,A -85,B 0,C 180,E1 -23305.105,E2 -23305.105} C_VEL
LIN {X 0,Y 165.293,Z 223.89,A -85,B 0,C 180,E1 -23309.998,E2 -23309.998} C_VEL
LIN {X 0,Y 164.77,Z 223.962,A -85,B 0,C 180,E1 -23314.892,E2 -23314.892} C_VEL
LIN {X 0,Y 164.848,Z 223.945,A -85,B 0,C 180,E1 -23317.346,E2 -23317.346} C_VEL
LIN {X 0,Y 164.75,Z 223.964,A -85,B 0,C 180,E1 -23321.15,E2 -23321.15} C_VEL
LIN {X 0,Y 164.481,Z 223.993,A -85,B 0,C 180,E1 -23327.401,E2 -23327.401} C_VEL
LIN {X 0,Y 164.469,Z 223.997,A -85,B 0,C 180,E1 -23329.988,E2 -23329.988} C_VEL
LIN {X 0,Y 164.389,Z 224.004,A -85,B 0,C 180,E1 -23336.133,E2 -23336.133} C_VEL
LIN {X 0,Y 164.371,Z 224.007,A -85,B 0,C 180,E1 -23341.227,E2 -23341.227} C_VEL
LIN {X 0,Y 164.342,Z 224.014,A -85,B 0,C 180,E1 -23346.774,E2 -23346.774} C_VEL
LIN {X 0,Y 164.363,Z 224.009,A -85,B 0,C 180,E1 -23349.893,E2 -23349.893} C_VEL
LIN {X 0,Y 164.373,Z 224.007,A -85,B 0,C 180,E1 -23353.378,E2 -23353.378} C_VEL
LIN {X 0,Y 164.372,Z 224.009,A -85,B 0,C 180,E1 -23356.836,E2 -23356.836} C_VEL
LIN {X 0,Y 164.333,Z 224.011,A -85,B 0,C 180,E1 -23360.333,E2 -23360.333} C_VEL
LIN {X 0,Y 164.338,Z 224.015,A -85,B 0,C 180,E1 -23364.341,E2 -23364.341} C_VEL
LIN {X 0,Y 164.384,Z 224.003,A -85,B 0,C 180,E1 -23369.135,E2 -23369.135} C_VEL
LIN {X 0,Y 164.41,Z 224.003,A -85,B 0,C 180,E1 -23374.694,E2 -23374.694} C_VEL
LIN {X 0,Y 164.478,Z 223.998,A -85,B 0,C 180,E1 -23380.051,E2 -23380.051} C_VEL
LIN {X 0,Y 164.499,Z 223.989,A -85,B 0,C 180,E1 -23385.148,E2 -23385.148} C_VEL
LIN {X 0,Y 164.762,Z 223.961,A -85,B 0,C 180,E1 -23390.177,E2 -23390.177} C_VEL
LIN {X 0,Y 164.825,Z 223.949,A -85,B 0,C 180,E1 -23392.652,E2 -23392.652} C_VEL
LIN {X 0,Y 165.041,Z 223.927,A -85,B 0,C 180,E1 -23397.561,E2 -23397.561} C_VEL
LIN {X 0,Y 165.289,Z 223.894,A -85,B 0,C 180,E1 -23400.001,E2 -23400.001} C_VEL
LIN {X 0,Y 164.767,Z 223.959,A -85,B 0,C 180,E1 -23404.895,E2 -23404.895} C_VEL
LIN {X 0,Y 164.849,Z 223.951,A -85,B 0,C 180,E1 -23407.349,E2 -23407.349} C_VEL
LIN {X 0,Y 164.738,Z 223.959,A -85,B 0,C 180,E1 -23411.133,E2 -23411.133} C_VEL
LIN {X 0,Y 164.479,Z 223.994,A -85,B 0,C 180,E1 -23417.405,E2 -23417.405} C_VEL
LIN {X 0,Y 164.469,Z 223.995,A -85,B 0,C 180,E1 -23419.991,E2 -23419.991} C_VEL
LIN {X 0,Y 164.389,Z 224.004,A -85,B 0,C 180,E1 -23426.135,E2 -23426.135} C_VEL
LIN {X 0,Y 164.37,Z 224.01,A -85,B 0,C 180,E1 -23431.229,E2 -23431.229} C_VEL
LIN {X 0,Y 164.291,Z 224.019,A -85,B 0,C 180,E1 -23436.792,E2 -23436.792} C_VEL
LIN {X 0,Y 164.288,Z 224.02,A -85,B 0,C 180,E1 -23439.918,E2 -23439.918} C_VEL
LIN {X 0,Y 164.277,Z 224.023,A -85,B 0,C 180,E1 -23443.344,E2 -23443.344} C_VEL
LIN {X 0,Y 164.328,Z 224.239,A -85,B 0,C 180,E1 -23446.994,E2 -23446.994} C_VEL
LIN {X 0,Y 166.636,Z 234.161,A -85,B 0,C 180,E1 -23451.571,E2 -23451.571} C_VEL
LIN {X 0,Y 169.164,Z 245.79,A -85,B 0,C 180,E1 -23456.583,E2 -23456.583} C_VEL
LIN {X 0,Y 170.003,Z 249.655,A -85,B 0,C 180,E1 -23458.193,E2 -23458.193} C_VEL
LIN {X 0,Y 170.128,Z 251.436,A -85,B 0,C 180,E1 -23458.913,E2 -23458.913} C_VEL
LIN {X 0,Y 169.714,Z 253.47,A -85,B 0,C 180,E1 -23459.605,E2 -23459.605} C_VEL
LIN {X 0,Y 169.916,Z 274.41,A -85,B 0,C 180,E1 -23460.924,E2 -23460.924} C_VEL
LIN {X 0,Y 171.599,Z 305.412,A -85,B 0,C 180,E1 -23462.896,E2 -23462.896} C_VEL
LIN {X 0,Y 169.591,Z 354.558,A -85,B 0,C 180,E1 -23465.854,E2 -23465.854} C_VEL
LIN {X 0,Y 168.798,Z 367.26,A -85,B 0,C 180,E1 -23467.085,E2 -23467.085} C_VEL
LIN {X 0,Y 167.646,Z 379.627,A -85,B 0,C 180,E1 -23468.805,E2 -23468.805} C_VEL
LIN {X 0,Y 166.459,Z 391.043,A -85,B 0,C 180,E1 -23470.903,E2 -23470.903} C_VEL
LIN {X 0,Y 165.198,Z 402.437,A -85,B 0,C 180,E1 -23473.631,E2 -23473.631} C_VEL
LIN {X 0,Y 164.359,Z 411.64,A -85,B 0,C 180,E1 -23476.4,E2 -23476.4} C_VEL
LIN {X 0,Y 163.89,Z 420.781,A -85,B 0,C 180,E1 -23479.851,E2 -23479.851} C_VEL
LIN {X 0,Y 163.229,Z 424.335,A -85,B 0,C 180,E1 -23481.485,E2 -23481.485} C_VEL
LIN {X 0,Y 161.721,Z 427.409,A -85,B 0,C 180,E1 -23483.198,E2 -23483.198} C_VEL
LIN {X 0,Y 158.265,Z 432.551,A -85,B 0,C 180,E1 -23486.89,E2 -23486.89} C_VEL
LIN {X 0,Y 157.297,Z 435.688,A -85,B 0,C 180,E1 -23489.542,E2 -23489.542} C_VEL
LIN {X 0,Y 156.931,Z 438.719,A -85,B 0,C 180,E1 -23492.569,E2 -23492.569} C_VEL
LIN {X 0,Y 155.957,Z 441.921,A -85,B 0,C 180,E1 -23497.511,E2 -23497.511} C_VEL
LIN {X 0,Y 155.831,Z 443.12,A -85,B 0,C 180,E1 -23500.395,E2 -23500.395} C_VEL
LIN {X 0,Y 156.825,Z 444.116,A -85,B 0,C 180,E1 -23505.6,E2 -23505.6} C_VEL
LIN {X 0,Y 159.416,Z 443.679,A -85,B 0,C 180,E1 -23510.653,E2 -23510.653} C_VEL
LIN {X 0,Y 163.44,Z 441.802,A -85,B 0,C 180,E1 -23515.469,E2 -23515.469} C_VEL
LIN {X 0,Y 168.793,Z 438.404,A -85,B 0,C 180,E1 -23519.978,E2 -23519.978} C_VEL
LIN {X 0,Y 173.739,Z 434.79,A -85,B 0,C 180,E1 -23523.101,E2 -23523.101} C_VEL
LIN {X 0,Y 179.37,Z 430.216,A -85,B 0,C 180,E1 -23525.997,E2 -23525.997} C_VEL
LIN {X 0,Y 186.697,Z 423.431,A -85,B 0,C 180,E1 -23529.091,E2 -23529.091} C_VEL
LIN {X 0,Y 194.641,Z 414.806,A -85,B 0,C 180,E1 -23531.913,E2 -23531.913} C_VEL
LIN {X 0,Y 200.79,Z 407.285,A -85,B 0,C 180,E1 -23533.733,E2 -23533.733} C_VEL
LIN {X 0,Y 207.282,Z 398.176,A -85,B 0,C 180,E1 -23535.4,E2 -23535.4} C_VEL
LIN {X 0,Y 214.103,Z 386.953,A -85,B 0,C 180,E1 -23536.918,E2 -23536.918} C_VEL
LIN {X 0,Y 219.743,Z 375.844,A -85,B 0,C 180,E1 -23538.04,E2 -23538.04} C_VEL
LIN {X 0,Y 224.932,Z 363.191,A -85,B 0,C 180,E1 -23538.992,E2 -23538.992} C_VEL
LIN {X 0,Y 229.107,Z 349.736,A -85,B 0,C 180,E1 -23539.702,E2 -23539.702} C_VEL
LIN {X 0,Y 232.643,Z 332.43,A -85,B 0,C 180,E1 -23540.406,E2 -23540.406} C_VEL
LIN {X 0,Y 233.388,Z 328.135,A -85,B 0,C 180,E1 -23540.621,E2 -23540.621} C_VEL
LIN {X 0,Y 232.923,Z 325.653,A -85,B 0,C 180,E1 -23542.07,E2 -23542.07} C_VEL
LIN {X 0,Y 232.293,Z 322.637,A -85,B 0,C 180,E1 -23544.91,E2 -23544.91} C_VEL
LIN {X 0,Y 232.222,Z 322.027,A -85,B 0,C 180,E1 -23545.861,E2 -23545.861} C_VEL
LIN {X 0,Y 232.399,Z 322.043,A -85,B 0,C 180,E1 -23549.427,E2 -23549.427} C_VEL
LIN {X 0,Y 233.179,Z 323.693,A -85,B 0,C 180,E1 -23552.068,E2 -23552.068} C_VEL
LIN {X 0,Y 233.511,Z 324.893,A -85,B 0,C 180,E1 -23553.039,E2 -23553.039} C_VEL
LIN {X 0,Y 229.81,Z 342.859,A -85,B 0,C 180,E1 -23553.937,E2 -23553.937} C_VEL
LIN {X 0,Y 226.366,Z 354.498,A -85,B 0,C 180,E1 -23554.781,E2 -23554.781} C_VEL
LIN {X 0,Y 221.751,Z 366.334,A -85,B 0,C 180,E1 -23555.917,E2 -23555.917} C_VEL
LIN {X 0,Y 216.046,Z 377.769,A -85,B 0,C 180,E1 -23557.381,E2 -23557.381} C_VEL
LIN {X 0,Y 209.394,Z 388.569,A -85,B 0,C 180,E1 -23559.261,E2 -23559.261} C_VEL
LIN {X 0,Y 202.759,Z 397.415,A -85,B 0,C 180,E1 -23561.298,E2 -23561.298} C_VEL
LIN {X 0,Y 196.735,Z 404.194,A -85,B 0,C 180,E1 -23563.393,E2 -23563.393} C_VEL
LIN {X 0,Y 189.825,Z 410.684,A -85,B 0,C 180,E1 -23566.074,E2 -23566.074} C_VEL
LIN {X 0,Y 183.477,Z 415.601,A -85,B 0,C 180,E1 -23568.957,E2 -23568.957} C_VEL
LIN {X 0,Y 176.789,Z 419.53,A -85,B 0,C 180,E1 -23572.561,E2 -23572.561} C_VEL
LIN {X 0,Y 172.458,Z 421.368,A -85,B 0,C 180,E1 -23575.324,E2 -23575.324} C_VEL
LIN {X 0,Y 168.774,Z 422.334,A -85,B 0,C 180,E1 -23578.042,E2 -23578.042} C_VEL
LIN {X 0,Y 163.966,Z 422.425,A -85,B 0,C 180,E1 -23582.455,E2 -23582.455} C_VEL
LIN {X 0,Y 161.782,Z 421.729,A -85,B 0,C 180,E1 -23584.983,E2 -23584.983} C_VEL
LIN {X 0,Y 159.966,Z 420.555,A -85,B 0,C 180,E1 -23587.573,E2 -23587.573} C_VEL
LIN {X 0,Y 157.8,Z 417.794,A -85,B 0,C 180,E1 -23591.524,E2 -23591.524} C_VEL
LIN {X 0,Y 156.302,Z 413.699,A -85,B 0,C 180,E1 -23595.65,E2 -23595.65} C_VEL
LIN {X 0,Y 155.671,Z 408.202,A -85,B 0,C 180,E1 -23599.789,E2 -23599.789} C_VEL
LIN {X 0,Y 155.715,Z 401.003,A -85,B 0,C 180,E1 -23603.965,E2 -23603.965} C_VEL
LIN {X 0,Y 156.234,Z 393.404,A -85,B 0,C 180,E1 -23607.456,E2 -23607.456} C_VEL
LIN {X 0,Y 156.994,Z 383.962,A -85,B 0,C 180,E1 -23610.931,E2 -23610.931} C_VEL
LIN {X 0,Y 158.044,Z 372.697,A -85,B 0,C 180,E1 -23614.152,E2 -23614.152} C_VEL
LIN {X 0,Y 159.123,Z 361.733,A -85,B 0,C 180,E1 -23616.601,E2 -23616.601} C_VEL
LIN {X 0,Y 160.207,Z 349.677,A -85,B 0,C 180,E1 -23618.69,E2 -23618.69} C_VEL
LIN {X 0,Y 161.159,Z 336.801,A -85,B 0,C 180,E1 -23620.338,E2 -23620.338} C_VEL
LIN {X 0,Y 161.818,Z 323.93,A -85,B 0,C 180,E1 -23621.47,E2 -23621.47} C_VEL
LIN {X 0,Y 164.494,Z 267.338,A -85,B 0,C 180,E1 -23625.28,E2 -23625.28} C_VEL
LIN {X 0,Y 162.036,Z 245.966,A -85,B 0,C 180,E1 -23626.911,E2 -23626.911} C_VEL
LIN {X 0,Y 160.206,Z 238.603,A -85,B 0,C 180,E1 -23627.628,E2 -23627.628} C_VEL
LIN {X 0,Y 157.864,Z 227.296,A -85,B 0,C 180,E1 -23633.257,E2 -23633.257} C_VEL
LIN {X 0,Y 157.414,Z 225.07,A -85,B 0,C 180,E1 -23634.519,E2 -23634.519} C_VEL
LIN {X 0,Y 157.28,Z 224.893,A -85,B 0,C 180,E1 -23640.557,E2 -23640.557} C_VEL
LIN {X 0,Y 157.322,Z 224.889,A -85,B 0,C 180,E1 -23643.464,E2 -23643.464} C_VEL
LIN {X 0,Y 157.393,Z 224.88,A -85,B 0,C 180,E1 -23649.665,E2 -23649.665} C_VEL
LIN {X 0,Y 157.461,Z 224.867,A -85,B 0,C 180,E1 -23654.465,E2 -23654.465} C_VEL
LIN {X 0,Y 157.769,Z 224.829,A -85,B 0,C 180,E1 -23659.734,E2 -23659.734} C_VEL
LIN {X 0,Y 157.82,Z 224.822,A -85,B 0,C 180,E1 -23662.321,E2 -23662.321} C_VEL
LIN {X 0,Y 158.256,Z 224.766,A -85,B 0,C 180,E1 -23669.998,E2 -23669.998} C_VEL
LIN {X 0,Y 157.806,Z 224.822,A -85,B 0,C 180,E1 -23677.676,E2 -23677.676} C_VEL
LIN {X 0,Y 157.679,Z 224.844,A -85,B 0,C 180,E1 -23681.319,E2 -23681.319} C_VEL
LIN {X 0,Y 157.458,Z 224.866,A -85,B 0,C 180,E1 -23685.532,E2 -23685.532} C_VEL
LIN {X 0,Y 157.366,Z 224.883,A -85,B 0,C 180,E1 -23690.931,E2 -23690.931} C_VEL
LIN {X 0,Y 157.31,Z 224.888,A -85,B 0,C 180,E1 -23696.684,E2 -23696.684} C_VEL
LIN {X 0,Y 157.272,Z 224.891,A -85,B 0,C 180,E1 -23702.426,E2 -23702.426} C_VEL
LIN {X 0,Y 157.317,Z 224.889,A -85,B 0,C 180,E1 -23706.475,E2 -23706.475} C_VEL
LIN {X 0,Y 157.281,Z 224.888,A -85,B 0,C 180,E1 -23712.084,E2 -23712.084} C_VEL
LIN {X 0,Y 157.293,Z 224.891,A -85,B 0,C 180,E1 -23715.631,E2 -23715.631} C_VEL
LIN {X 0,Y 157.26,Z 224.892,A -85,B 0,C 180,E1 -23721.271,E2 -23721.271} C_VEL
LIN {X 0,Y 157.286,Z 224.893,A -85,B 0,C 180,E1 -23724.489,E2 -23724.489} C_VEL
LIN {X 0,Y 157.288,Z 224.888,A -85,B 0,C 180,E1 -23728.095,E2 -23728.095} C_VEL
LIN {X 0,Y 157.315,Z 224.888,A -85,B 0,C 180,E1 -23733.466,E2 -23733.466} C_VEL
LIN {X 0,Y 157.387,Z 224.879,A -85,B 0,C 180,E1 -23739.668,E2 -23739.668} C_VEL
LIN {X 0,Y 157.436,Z 224.869,A -85,B 0,C 180,E1 -23744.465,E2 -23744.465} C_VEL
LIN {X 0,Y 157.683,Z 224.844,A -85,B 0,C 180,E1 -23749.732,E2 -23749.732} C_VEL
LIN {X 0,Y 157.761,Z 224.829,A -85,B 0,C 180,E1 -23752.321,E2 -23752.321} C_VEL
LIN {X 0,Y 158.251,Z 224.77,A -85,B 0,C 180,E1 -23760.001,E2 -23760.001} C_VEL
LIN {X 0,Y 157.805,Z 224.828,A -85,B 0,C 180,E1 -23767.679,E2 -23767.679} C_VEL
LIN {X 0,Y 157.668,Z 224.84,A -85,B 0,C 180,E1 -23771.304,E2 -23771.304} C_VEL
LIN {X 0,Y 157.45,Z 224.873,A -85,B 0,C 180,E1 -23775.536,E2 -23775.536} C_VEL
LIN {X 0,Y 157.366,Z 224.88,A -85,B 0,C 180,E1 -23780.935,E2 -23780.935} C_VEL
LIN {X 0,Y 157.31,Z 224.886,A -85,B 0,C 180,E1 -23786.686,E2 -23786.686} C_VEL
LIN {X 0,Y 157.271,Z 224.892,A -85,B 0,C 180,E1 -23792.43,E2 -23792.43} C_VEL
LIN {X 0,Y 157.265,Z 224.894,A -85,B 0,C 180,E1 -23796.451,E2 -23796.451} C_VEL
LIN {X 0,Y 157.19,Z 224.905,A -85,B 0,C 180,E1 -23802.119,E2 -23802.119} C_VEL
LIN {X 0,Y 157.279,Z 225.098,A -85,B 0,C 180,E1 -23806.435,E2 -23806.435} C_VEL
LIN {X 0,Y 159.587,Z 235.106,A -85,B 0,C 180,E1 -23811.248,E2 -23811.248} C_VEL
LIN {X 0,Y 162.508,Z 248.575,A -85,B 0,C 180,E1 -23817.279,E2 -23817.279} C_VEL
LIN {X 0,Y 162.926,Z 250.478,A -85,B 0,C 180,E1 -23818.104,E2 -23818.104} C_VEL
LIN {X 0,Y 162.798,Z 252.927,A -85,B 0,C 180,E1 -23819.053,E2 -23819.053} C_VEL
LIN {X 0,Y 162.652,Z 265.704,A -85,B 0,C 180,E1 -23819.941,E2 -23819.941} C_VEL
LIN {X 0,Y 164.572,Z 305.456,A -85,B 0,C 180,E1 -23822.589,E2 -23822.589} C_VEL
LIN {X 0,Y 162.514,Z 354.321,A -85,B 0,C 180,E1 -23825.71,E2 -23825.71} C_VEL
LIN {X 0,Y 161.737,Z 366.731,A -85,B 0,C 180,E1 -23826.98,E2 -23826.98} C_VEL
LIN {X 0,Y 160.535,Z 379.393,A -85,B 0,C 180,E1 -23828.83,E2 -23828.83} C_VEL
LIN {X 0,Y 159.355,Z 390.713,A -85,B 0,C 180,E1 -23831.021,E2 -23831.021} C_VEL
LIN {X 0,Y 158.124,Z 402.055,A -85,B 0,C 180,E1 -23833.874,E2 -23833.874} C_VEL
LIN {X 0,Y 157.3,Z 412.103,A -85,B 0,C 180,E1 -23837.093,E2 -23837.093} C_VEL
LIN {X 0,Y 156.919,Z 420.562,A -85,B 0,C 180,E1 -23840.488,E2 -23840.488} C_VEL
LIN {X 0,Y 156.918,Z 427.944,A -85,B 0,C 180,E1 -23844.218,E2 -23844.218} C_VEL
LIN {X 0,Y 157.148,Z 433.012,A -85,B 0,C 180,E1 -23847.439,E2 -23847.439} C_VEL
LIN {X 0,Y 157.297,Z 435.688,A -85,B 0,C 180,E1 -23849.542,E2 -23849.542} C_VEL
LIN {X 0,Y 156.943,Z 437.078,A -85,B 0,C 180,E1 -23850.869,E2 -23850.869} C_VEL
LIN {X 0,Y 155.334,Z 438.596,A -85,B 0,C 180,E1 -23852.875,E2 -23852.875} C_VEL
LIN {X 0,Y 150.181,Z 440.749,A -85,B 0,C 180,E1 -23857.739,E2 -23857.739} C_VEL
LIN {X 0,Y 148.978,Z 441.52,A -85,B 0,C 180,E1 -23859.991,E2 -23859.991} C_VEL
LIN {X 0,Y 148.906,Z 441.783,A -85,B 0,C 180,E1 -23860.756,E2 -23860.756} C_VEL
LIN {X 0,Y 150.021,Z 443.135,A -85,B 0,C 180,E1 -23866.326,E2 -23866.326} C_VEL
LIN {X 0,Y 152.772,Z 443.025,A -85,B 0,C 180,E1 -23871.596,E2 -23871.596} C_VEL
LIN {X 0,Y 157.032,Z 441.452,A -85,B 0,C 180,E1 -23876.588,E2 -23876.588} C_VEL
LIN {X 0,Y 162.671,Z 438.45,A -85,B 0,C 180,E1 -23881.23,E2 -23881.23} C_VEL
LIN {X 0,Y 167.857,Z 435.175,A -85,B 0,C 180,E1 -23884.42,E2 -23884.42} C_VEL
LIN {X 0,Y 173.709,Z 430.919,A -85,B 0,C 180,E1 -23887.366,E2 -23887.366} C_VEL
LIN {X 0,Y 182.432,Z 423.55,A -85,B 0,C 180,E1 -23890.914,E2 -23890.914} C_VEL
LIN {X 0,Y 189.529,Z 416.585,A -85,B 0,C 180,E1 -23893.316,E2 -23893.316} C_VEL
LIN {X 0,Y 197.132,Z 407.936,A -85,B 0,C 180,E1 -23895.483,E2 -23895.483} C_VEL
LIN {X 0,Y 203.862,Z 399.229,A -85,B 0,C 180,E1 -23897.104,E2 -23897.104} C_VEL
LIN {X 0,Y 210.904,Z 388.564,A -85,B 0,C 180,E1 -23898.572,E2 -23898.572} C_VEL
LIN {X 0,Y 216.972,Z 377.494,A -85,B 0,C 180,E1 -23899.714,E2 -23899.714} C_VEL
LIN {X 0,Y 222.426,Z 365.135,A -85,B 0,C 180,E1 -23900.634,E2 -23900.634} C_VEL
LIN {X 0,Y 226.86,Z 352.304,A -85,B 0,C 180,E1 -23901.338,E2 -23901.338} C_VEL
LIN {X 0,Y 230.31,Z 338.17,A -85,B 0,C 180,E1 -23901.925,E2 -23901.925} C_VEL
LIN {X 0,Y 231.329,Z 332.737,A -85,B 0,C 180,E1 -23902.178,E2 -23902.178} C_VEL
LIN {X 0,Y 230.748,Z 329.463,A -85,B 0,C 180,E1 -23905.195,E2 -23905.195} C_VEL
LIN {X 0,Y 230.628,Z 328.804,A -85,B 0,C 180,E1 -23906.734,E2 -23906.734} C_VEL
LIN {X 0,Y 230.912,Z 329.023,A -85,B 0,C 180,E1 -23909.606,E2 -23909.606} C_VEL
LIN {X 0,Y 231.399,Z 330.462,A -85,B 0,C 180,E1 -23911.565,E2 -23911.565} C_VEL
LIN {X 0,Y 228.278,Z 344.386,A -85,B 0,C 180,E1 -23912.243,E2 -23912.243} C_VEL
LIN {X 0,Y 224.106,Z 357.308,A -85,B 0,C 180,E1 -23913.193,E2 -23913.193} C_VEL
LIN {X 0,Y 218.866,Z 369.4,A -85,B 0,C 180,E1 -23914.379,E2 -23914.379} C_VEL
LIN {X 0,Y 213.42,Z 379.597,A -85,B 0,C 180,E1 -23915.692,E2 -23915.692} C_VEL
LIN {X 0,Y 207.505,Z 388.725,A -85,B 0,C 180,E1 -23917.241,E2 -23917.241} C_VEL
LIN {X 0,Y 201.241,Z 396.817,A -85,B 0,C 180,E1 -23919.023,E2 -23919.023} C_VEL
LIN {X 0,Y 194.815,Z 403.879,A -85,B 0,C 180,E1 -23921.053,E2 -23921.053} C_VEL
LIN {X 0,Y 187.411,Z 410.662,A -85,B 0,C 180,E1 -23923.664,E2 -23923.664} C_VEL
LIN {X 0,Y 180.511,Z 415.739,A -85,B 0,C 180,E1 -23926.49,E2 -23926.49} C_VEL
LIN {X 0,Y 174.192,Z 419.496,A -85,B 0,C 180,E1 -23929.538,E2 -23929.538} C_VEL
LIN {X 0,Y 168.498,Z 421.931,A -85,B 0,C 180,E1 -23932.811,E2 -23932.811} C_VEL
LIN {X 0,Y 165,Z 422.893,A -85,B 0,C 180,E1 -23935.112,E2 -23935.112} C_VEL
LIN {X 0,Y 161.8,Z 423.389,A -85,B 0,C 180,E1 -23937.509,E2 -23937.509} C_VEL
LIN {X 0,Y 158.958,Z 423.335,A -85,B 0,C 180,E1 -23939.999,E2 -23939.999} C_VEL
LIN {X 0,Y 155.035,Z 422.223,A -85,B 0,C 180,E1 -23944.199,E2 -23944.199} C_VEL
LIN {X 0,Y 151.652,Z 419.193,A -85,B 0,C 180,E1 -23949.333,E2 -23949.333} C_VEL
LIN {X 0,Y 149.85,Z 415.404,A -85,B 0,C 180,E1 -23953.561,E2 -23953.561} C_VEL
LIN {X 0,Y 148.813,Z 410.428,A -85,B 0,C 180,E1 -23957.728,E2 -23957.728} C_VEL
LIN {X 0,Y 148.544,Z 404.732,A -85,B 0,C 180,E1 -23961.509,E2 -23961.509} C_VEL
LIN {X 0,Y 148.805,Z 397.894,A -85,B 0,C 180,E1 -23965.153,E2 -23965.153} C_VEL
LIN {X 0,Y 149.42,Z 389.319,A -85,B 0,C 180,E1 -23968.822,E2 -23968.822} C_VEL
LIN {X 0,Y 150.235,Z 379.733,A -85,B 0,C 180,E1 -23972.11,E2 -23972.11} C_VEL
LIN {X 0,Y 151.315,Z 368.866,A -85,B 0,C 180,E1 -23975.082,E2 -23975.082} C_VEL
LIN {X 0,Y 152.53,Z 356.302,A -85,B 0,C 180,E1 -23977.735,E2 -23977.735} C_VEL
LIN {X 0,Y 153.672,Z 342.898,A -85,B 0,C 180,E1 -23979.81,E2 -23979.81} C_VEL
LIN {X 0,Y 154.504,Z 329.464,A -85,B 0,C 180,E1 -23981.265,E2 -23981.265} C_VEL
LIN {X 0,Y 157.501,Z 268.006,A -85,B 0,C 180,E1 -23985.638,E2 -23985.638} C_VEL
LIN {X 0,Y 155.105,Z 247.291,A -85,B 0,C 180,E1 -23987.296,E2 -23987.296} C_VEL
LIN {X 0,Y 153.028,Z 238.953,A -85,B 0,C 180,E1 -23988.136,E2 -23988.136} C_VEL
LIN {X 0,Y 150.882,Z 228.485,A -85,B 0,C 180,E1 -23993.565,E2 -23993.565} C_VEL
LIN {X 0,Y 150.342,Z 225.862,A -85,B 0,C 180,E1 -23995.165,E2 -23995.165} C_VEL
LIN {X 0,Y 150.217,Z 225.774,A -85,B 0,C 180,E1 -23999.025,E2 -23999.025} C_VEL
LIN {X 0,Y 150.245,Z 225.769,A -85,B 0,C 180,E1 -24002.715,E2 -24002.715} C_VEL
LIN {X 0,Y 150.35,Z 225.757,A -85,B 0,C 180,E1 -24009.205,E2 -24009.205} C_VEL
LIN {X 0,Y 150.367,Z 225.751,A -85,B 0,C 180,E1 -24013.712,E2 -24013.712} C_VEL
LIN {X 0,Y 150.686,Z 225.713,A -85,B 0,C 180,E1 -24019.246,E2 -24019.246} C_VEL
LIN {X 0,Y 150.759,Z 225.701,A -85,B 0,C 180,E1 -24021.959,E2 -24021.959} C_VEL
LIN {X 0,Y 151.216,Z 225.643,A -85,B 0,C 180,E1 -24029.998,E2 -24029.998} C_VEL
LIN {X 0,Y 150.741,Z 225.701,A -85,B 0,C 180,E1 -24038.038,E2 -24038.038} C_VEL
LIN {X 0,Y 150.61,Z 225.724,A -85,B 0,C 180,E1 -24041.505,E2 -24041.505} C_VEL
LIN {X 0,Y 150.364,Z 225.75,A -85,B 0,C 180,E1 -24046.284,E2 -24046.284} C_VEL
LIN {X 0,Y 150.347,Z 225.758,A -85,B 0,C 180,E1 -24050.791,E2 -24050.791} C_VEL
LIN {X 0,Y 150.24,Z 225.769,A -85,B 0,C 180,E1 -24057.281,E2 -24057.281} C_VEL
LIN {X 0,Y 150.213,Z 225.769,A -85,B 0,C 180,E1 -24062.633,E2 -24062.633} C_VEL
LIN {X 0,Y 150.227,Z 225.771,A -85,B 0,C 180,E1 -24067.455,E2 -24067.455} C_VEL
LIN {X 0,Y 150.222,Z 225.766,A -85,B 0,C 180,E1 -24071.538,E2 -24071.538} C_VEL
LIN {X 0,Y 150.243,Z 225.769,A -85,B 0,C 180,E1 -24075.442,E2 -24075.442} C_VEL
LIN {X 0,Y 150.201,Z 225.77,A -85,B 0,C 180,E1 -24079.077,E2 -24079.077} C_VEL
LIN {X 0,Y 150.222,Z 225.772,A -85,B 0,C 180,E1 -24082.682,E2 -24082.682} C_VEL
LIN {X 0,Y 150.212,Z 225.77,A -85,B 0,C 180,E1 -24087.365,E2 -24087.365} C_VEL
LIN {X 0,Y 150.238,Z 225.77,A -85,B 0,C 180,E1 -24092.718,E2 -24092.718} C_VEL
LIN {X 0,Y 150.345,Z 225.755,A -85,B 0,C 180,E1 -24099.208,E2 -24099.208} C_VEL
LIN {X 0,Y 150.347,Z 225.755,A -85,B 0,C 180,E1 -24103.713,E2 -24103.713} C_VEL
LIN {X 0,Y 150.605,Z 225.724,A -85,B 0,C 180,E1 -24109.243,E2 -24109.243} C_VEL
LIN {X 0,Y 150.699,Z 225.71,A -85,B 0,C 180,E1 -24111.959,E2 -24111.959} C_VEL
LIN {X 0,Y 151.212,Z 225.647,A -85,B 0,C 180,E1 -24120.001,E2 -24120.001} C_VEL
LIN {X 0,Y 150.739,Z 225.706,A -85,B 0,C 180,E1 -24128.042,E2 -24128.042} C_VEL
LIN {X 0,Y 150.602,Z 225.721,A -85,B 0,C 180,E1 -24131.494,E2 -24131.494} C_VEL
LIN {X 0,Y 150.357,Z 225.754,A -85,B 0,C 180,E1 -24136.288,E2 -24136.288} C_VEL
LIN {X 0,Y 150.347,Z 225.754,A -85,B 0,C 180,E1 -24140.794,E2 -24140.794} C_VEL
LIN {X 0,Y 150.24,Z 225.766,A -85,B 0,C 180,E1 -24147.284,E2 -24147.284} C_VEL
LIN {X 0,Y 150.211,Z 225.772,A -85,B 0,C 180,E1 -24152.634,E2 -24152.634} C_VEL
LIN {X 0,Y 150.17,Z 225.78,A -85,B 0,C 180,E1 -24157.476,E2 -24157.476} C_VEL
LIN {X 0,Y 150.134,Z 225.785,A -85,B 0,C 180,E1 -24161.501,E2 -24161.501} C_VEL
LIN {X 0,Y 150.211,Z 226.014,A -85,B 0,C 180,E1 -24165.866,E2 -24165.866} C_VEL
LIN {X 0,Y 152.498,Z 235.997,A -85,B 0,C 180,E1 -24170.894,E2 -24170.894} C_VEL
LIN {X 0,Y 155.081,Z 247.64,A -85,B 0,C 180,E1 -24176.372,E2 -24176.372} C_VEL
LIN {X 0,Y 155.849,Z 252.603,A -85,B 0,C 180,E1 -24178.567,E2 -24178.567} C_VEL
LIN {X 0,Y 155.752,Z 269.844,A -85,B 0,C 180,E1 -24179.794,E2 -24179.794} C_VEL
LIN {X 0,Y 157.492,Z 306.122,A -85,B 0,C 180,E1 -24182.333,E2 -24182.333} C_VEL
LIN {X 0,Y 155.481,Z 353.77,A -85,B 0,C 180,E1 -24185.534,E2 -24185.534} C_VEL
LIN {X 0,Y 154.741,Z 365.349,A -85,B 0,C 180,E1 -24186.763,E2 -24186.763} C_VEL
LIN {X 0,Y 153.624,Z 377.319,A -85,B 0,C 180,E1 -24188.534,E2 -24188.534} C_VEL
LIN {X 0,Y 152.427,Z 388.945,A -85,B 0,C 180,E1 -24190.824,E2 -24190.824} C_VEL
LIN {X 0,Y 151.29,Z 399.38,A -85,B 0,C 180,E1 -24193.471,E2 -24193.471} C_VEL
LIN {X 0,Y 150.417,Z 408.848,A -85,B 0,C 180,E1 -24196.492,E2 -24196.492} C_VEL
LIN {X 0,Y 149.991,Z 417.087,A -85,B 0,C 180,E1 -24199.736,E2 -24199.736} C_VEL
LIN {X 0,Y 149.908,Z 424.321,A -85,B 0,C 180,E1 -24203.271,E2 -24203.271} C_VEL
LIN {X 0,Y 150.079,Z 428.903,A -85,B 0,C 180,E1 -24205.974,E2 -24205.974} C_VEL
LIN {X 0,Y 150.42,Z 434.198,A -85,B 0,C 180,E1 -24209.865,E2 -24209.865} C_VEL
LIN {X 0,Y 150.031,Z 437.002,A -85,B 0,C 180,E1 -24212.687,E2 -24212.687} C_VEL
LIN {X 0,Y 148.99,Z 440.518,A -85,B 0,C 180,E1 -24217.858,E2 -24217.858} C_VEL
LIN {X 0,Y 148.906,Z 441.783,A -85,B 0,C 180,E1 -24220.756,E2 -24220.756} C_VEL
LIN {X 0,Y 148.474,Z 442.509,A -85,B 0,C 180,E1 -24223.011,E2 -24223.011} C_VEL
LIN {X 0,Y 146.617,Z 442.87,A -85,B 0,C 180,E1 -24226.794,E2 -24226.794} C_VEL
LIN {X 0,Y 145.585,Z 442.551,A -85,B 0,C 180,E1 -24230.657,E2 -24230.657} C_VEL
LIN {X 0,Y 146.431,Z 442.211,A -85,B 0,C 180,E1 -24232.944,E2 -24232.944} C_VEL
LIN {X 0,Y 150.694,Z 441.065,A -85,B 0,C 180,E1 -24237.801,E2 -24237.801} C_VEL
LIN {X 0,Y 156.644,Z 438.408,A -85,B 0,C 180,E1 -24242.576,E2 -24242.576} C_VEL
LIN {X 0,Y 164.002,Z 434.242,A -85,B 0,C 180,E1 -24246.867,E2 -24246.867} C_VEL
LIN {X 0,Y 170.33,Z 430.027,A -85,B 0,C 180,E1 -24249.76,E2 -24249.76} C_VEL
LIN {X 0,Y 178.391,Z 423.718,A -85,B 0,C 180,E1 -24252.813,E2 -24252.813} C_VEL
LIN {X 0,Y 185.791,Z 416.966,A -85,B 0,C 180,E1 -24255.177,E2 -24255.177} C_VEL
LIN {X 0,Y 193.684,Z 408.776,A -85,B 0,C 180,E1 -24257.291,E2 -24257.291} C_VEL
LIN {X 0,Y 200.635,Z 400.379,A -85,B 0,C 180,E1 -24258.863,E2 -24258.863} C_VEL
LIN {X 0,Y 207.864,Z 390.144,A -85,B 0,C 180,E1 -24260.282,E2 -24260.282} C_VEL
LIN {X 0,Y 214.421,Z 379.135,A -85,B 0,C 180,E1 -24261.429,E2 -24261.429} C_VEL
LIN {X 0,Y 220.114,Z 367.483,A -85,B 0,C 180,E1 -24262.298,E2 -24262.298} C_VEL
LIN {X 0,Y 224.699,Z 355.472,A -85,B 0,C 180,E1 -24262.98,E2 -24262.98} C_VEL
LIN {X 0,Y 228.493,Z 342.041,A -85,B 0,C 180,E1 -24263.549,E2 -24263.549} C_VEL
LIN {X 0,Y 229.35,Z 338.007,A -85,B 0,C 180,E1 -24263.736,E2 -24263.736} C_VEL
LIN {X 0,Y 229.185,Z 335.85,A -85,B 0,C 180,E1 -24266.131,E2 -24266.131} C_VEL
LIN {X 0,Y 229.353,Z 335.914,A -85,B 0,C 180,E1 -24269.378,E2 -24269.378} C_VEL
LIN {X 0,Y 229.418,Z 336.306,A -85,B 0,C 180,E1 -24270.041,E2 -24270.041} C_VEL
LIN {X 0,Y 226.368,Z 347.974,A -85,B 0,C 180,E1 -24270.656,E2 -24270.656} C_VEL
LIN {X 0,Y 222.347,Z 359.478,A -85,B 0,C 180,E1 -24271.518,E2 -24271.518} C_VEL
LIN {X 0,Y 217.369,Z 370.448,A -85,B 0,C 180,E1 -24272.565,E2 -24272.565} C_VEL
LIN {X 0,Y 211.305,Z 381.079,A -85,B 0,C 180,E1 -24273.901,E2 -24273.901} C_VEL
LIN {X 0,Y 204.274,Z 391.176,A -85,B 0,C 180,E1 -24275.615,E2 -24275.615} C_VEL
LIN {X 0,Y 197.45,Z 399.326,A -85,B 0,C 180,E1 -24277.446,E2 -24277.446} C_VEL
LIN {X 0,Y 190.611,Z 406.178,A -85,B 0,C 180,E1 -24279.495,E2 -24279.495} C_VEL
LIN {X 0,Y 182.854,Z 412.579,A -85,B 0,C 180,E1 -24282.092,E2 -24282.092} C_VEL
LIN {X 0,Y 176.042,Z 417.183,A -85,B 0,C 180,E1 -24284.737,E2 -24284.737} C_VEL
LIN {X 0,Y 168.964,Z 420.865,A -85,B 0,C 180,E1 -24287.995,E2 -24287.995} C_VEL
LIN {X 0,Y 163.737,Z 422.86,A -85,B 0,C 180,E1 -24290.835,E2 -24290.835} C_VEL
LIN {X 0,Y 157.494,Z 424.162,A -85,B 0,C 180,E1 -24294.878,E2 -24294.878} C_VEL
LIN {X 0,Y 154.27,Z 424.242,A -85,B 0,C 180,E1 -24297.388,E2 -24297.388} C_VEL
LIN {X 0,Y 151.401,Z 423.814,A -85,B 0,C 180,E1 -24299.999,E2 -24299.999} C_VEL
LIN {X 0,Y 147.927,Z 422.354,A -85,B 0,C 180,E1 -24303.861,E2 -24303.861} C_VEL
LIN {X 0,Y 144.934,Z 419.516,A -85,B 0,C 180,E1 -24308.363,E2 -24308.363} C_VEL
LIN {X 0,Y 142.975,Z 415.54,A -85,B 0,C 180,E1 -24312.777,E2 -24312.777} C_VEL
LIN {X 0,Y 141.796,Z 410.184,A -85,B 0,C 180,E1 -24317.299,E2 -24317.299} C_VEL
LIN {X 0,Y 141.507,Z 403.225,A -85,B 0,C 180,E1 -24321.868,E2 -24321.868} C_VEL
LIN {X 0,Y 141.849,Z 395.99,A -85,B 0,C 180,E1 -24325.69,E2 -24325.69} C_VEL
LIN {X 0,Y 142.368,Z 388.612,A -85,B 0,C 180,E1 -24328.842,E2 -24328.842} C_VEL
LIN {X 0,Y 143.192,Z 378.782,A -85,B 0,C 180,E1 -24332.258,E2 -24332.258} C_VEL
LIN {X 0,Y 144.244,Z 368.369,A -85,B 0,C 180,E1 -24335.151,E2 -24335.151} C_VEL
LIN {X 0,Y 145.429,Z 356.099,A -85,B 0,C 180,E1 -24337.815,E2 -24337.815} C_VEL
LIN {X 0,Y 146.497,Z 343.552,A -85,B 0,C 180,E1 -24339.861,E2 -24339.861} C_VEL
LIN {X 0,Y 147.364,Z 330.33,A -85,B 0,C 180,E1 -24341.387,E2 -24341.387} C_VEL
LIN {X 0,Y 150.381,Z 267.768,A -85,B 0,C 180,E1 -24346.1,E2 -24346.1} C_VEL
LIN {X 0,Y 148.169,Z 248.41,A -85,B 0,C 180,E1 -24347.714,E2 -24347.714} C_VEL
LIN {X 0,Y 145.874,Z 239.495,A -85,B 0,C 180,E1 -24348.627,E2 -24348.627} C_VEL
LIN {X 0,Y 144.101,Z 230.668,A -85,B 0,C 180,E1 -24353.311,E2 -24353.311} C_VEL
LIN {X 0,Y 143.338,Z 227.05,A -85,B 0,C 180,E1 -24355.403,E2 -24355.403} C_VEL
LIN {X 0,Y 143.24,Z 226.648,A -85,B 0,C 180,E1 -24356.09,E2 -24356.09} C_VEL
LIN {X 0,Y 143.192,Z 226.648,A -85,B 0,C 180,E1 -24362.059,E2 -24362.059} C_VEL
LIN {X 0,Y 143.276,Z 226.636,A -85,B 0,C 180,E1 -24368.743,E2 -24368.743} C_VEL
LIN {X 0,Y 143.304,Z 226.631,A -85,B 0,C 180,E1 -24372.885,E2 -24372.885} C_VEL
LIN {X 0,Y 143.6,Z 226.597,A -85,B 0,C 180,E1 -24378.709,E2 -24378.709} C_VEL
LIN {X 0,Y 143.681,Z 226.583,A -85,B 0,C 180,E1 -24381.56,E2 -24381.56} C_VEL
LIN {X 0,Y 144.175,Z 226.52,A -85,B 0,C 180,E1 -24389.998,E2 -24389.998} C_VEL
LIN {X 0,Y 143.662,Z 226.583,A -85,B 0,C 180,E1 -24398.437,E2 -24398.437} C_VEL
LIN {X 0,Y 143.544,Z 226.604,A -85,B 0,C 180,E1 -24401.711,E2 -24401.711} C_VEL
LIN {X 0,Y 143.301,Z 226.63,A -85,B 0,C 180,E1 -24407.111,E2 -24407.111} C_VEL
LIN {X 0,Y 143.272,Z 226.638,A -85,B 0,C 180,E1 -24411.253,E2 -24411.253} C_VEL
LIN {X 0,Y 143.186,Z 226.648,A -85,B 0,C 180,E1 -24417.936,E2 -24417.936} C_VEL
LIN {X 0,Y 143.163,Z 226.645,A -85,B 0,C 180,E1 -24423.434,E2 -24423.434} C_VEL
LIN {X 0,Y 143.118,Z 226.655,A -85,B 0,C 180,E1 -24429.668,E2 -24429.668} C_VEL
LIN {X 0,Y 143.155,Z 226.65,A -85,B 0,C 180,E1 -24433.414,E2 -24433.414} C_VEL
LIN {X 0,Y 143.141,Z 226.653,A -85,B 0,C 180,E1 -24437.429,E2 -24437.429} C_VEL
LIN {X 0,Y 143.121,Z 226.654,A -85,B 0,C 180,E1 -24441.78,E2 -24441.78} C_VEL
LIN {X 0,Y 143.18,Z 226.646,A -85,B 0,C 180,E1 -24447.322,E2 -24447.322} C_VEL
LIN {X 0,Y 143.184,Z 226.65,A -85,B 0,C 180,E1 -24452.063,E2 -24452.063} C_VEL
LIN {X 0,Y 143.27,Z 226.636,A -85,B 0,C 180,E1 -24458.746,E2 -24458.746} C_VEL
LIN {X 0,Y 143.29,Z 226.634,A -85,B 0,C 180,E1 -24462.887,E2 -24462.887} C_VEL
LIN {X 0,Y 143.531,Z 226.605,A -85,B 0,C 180,E1 -24468.706,E2 -24468.706} C_VEL
LIN {X 0,Y 143.62,Z 226.594,A -85,B 0,C 180,E1 -24471.56,E2 -24471.56} C_VEL
LIN {X 0,Y 144.171,Z 226.524,A -85,B 0,C 180,E1 -24480.001,E2 -24480.001} C_VEL
LIN {X 0,Y 143.658,Z 226.588,A -85,B 0,C 180,E1 -24488.441,E2 -24488.441} C_VEL
LIN {X 0,Y 143.543,Z 226.601,A -85,B 0,C 180,E1 -24491.714,E2 -24491.714} C_VEL
LIN {X 0,Y 143.297,Z 226.634,A -85,B 0,C 180,E1 -24497.115,E2 -24497.115} C_VEL
LIN {X 0,Y 143.273,Z 226.637,A -85,B 0,C 180,E1 -24501.257,E2 -24501.257} C_VEL
LIN {X 0,Y 143.187,Z 226.646,A -85,B 0,C 180,E1 -24507.939,E2 -24507.939} C_VEL
LIN {X 0,Y 143.14,Z 226.654,A -85,B 0,C 180,E1 -24513.422,E2 -24513.422} C_VEL
LIN {X 0,Y 143.053,Z 226.666,A -85,B 0,C 180,E1 -24519.695,E2 -24519.695} C_VEL
LIN {X 0,Y 143.137,Z 226.831,A -85,B 0,C 180,E1 -24525.233,E2 -24525.233} C_VEL
LIN {X 0,Y 145.461,Z 237.04,A -85,B 0,C 180,E1 -24530.63,E2 -24530.63} C_VEL
LIN {X 0,Y 148.307,Z 249.831,A -85,B 0,C 180,E1 -24536.915,E2 -24536.915} C_VEL
LIN {X 0,Y 148.818,Z 252.56,A -85,B 0,C 180,E1 -24538.099,E2 -24538.099} C_VEL
LIN {X 0,Y 148.907,Z 274.658,A -85,B 0,C 180,E1 -24539.71,E2 -24539.71} C_VEL
LIN {X 0,Y 150.5,Z 305.551,A -85,B 0,C 180,E1 -24541.975,E2 -24541.975} C_VEL
LIN {X 0,Y 148.426,Z 353.06,A -85,B 0,C 180,E1 -24545.34,E2 -24545.34} C_VEL
LIN {X 0,Y 147.656,Z 365.113,A -85,B 0,C 180,E1 -24546.696,E2 -24546.696} C_VEL
LIN {X 0,Y 146.531,Z 376.889,A -85,B 0,C 180,E1 -24548.551,E2 -24548.551} C_VEL
LIN {X 0,Y 145.344,Z 388.402,A -85,B 0,C 180,E1 -24550.952,E2 -24550.952} C_VEL
LIN {X 0,Y 144.242,Z 398.76,A -85,B 0,C 180,E1 -24553.732,E2 -24553.732} C_VEL
LIN {X 0,Y 143.385,Z 409.163,A -85,B 0,C 180,E1 -24557.26,E2 -24557.26} C_VEL
LIN {X 0,Y 143.046,Z 417.685,A -85,B 0,C 180,E1 -24560.905,E2 -24560.905} C_VEL
LIN {X 0,Y 143.158,Z 425.465,A -85,B 0,C 180,E1 -24565.074,E2 -24565.074} C_VEL
LIN {X 0,Y 143.437,Z 430.654,A -85,B 0,C 180,E1 -24568.598,E2 -24568.598} C_VEL
LIN {X 0,Y 143.458,Z 433.93,A -85,B 0,C 180,E1 -24571.406,E2 -24571.406} C_VEL
LIN {X 0,Y 142.471,Z 437.405,A -85,B 0,C 180,E1 -24575.664,E2 -24575.664} C_VEL
LIN {X 0,Y 142.004,Z 440.473,A -85,B 0,C 180,E1 -24581.42,E2 -24581.42} C_VEL
LIN {X 0,Y 143.244,Z 442.089,A -85,B 0,C 180,E1 -24587.122,E2 -24587.122} C_VEL
LIN {X 0,Y 146.193,Z 442.263,A -85,B 0,C 180,E1 -24592.62,E2 -24592.62} C_VEL
LIN {X 0,Y 146.431,Z 442.211,A -85,B 0,C 180,E1 -24592.944,E2 -24592.944} C_VEL
LIN {X 0,Y 147.539,Z 441.821,A -85,B 0,C 180,E1 -24595.203,E2 -24595.203} C_VEL
LIN {X 0,Y 148.173,Z 440.663,A -85,B 0,C 180,E1 -24599.02,E2 -24599.02} C_VEL
LIN {X 0,Y 149.582,Z 439.035,A -85,B 0,C 180,E1 -24602.732,E2 -24602.732} C_VEL
LIN {X 0,Y 151.825,Z 437.782,A -85,B 0,C 180,E1 -24604.742,E2 -24604.742} C_VEL
LIN {X 0,Y 158.401,Z 434.568,A -85,B 0,C 180,E1 -24608.402,E2 -24608.402} C_VEL
LIN {X 0,Y 164.962,Z 430.694,A -85,B 0,C 180,E1 -24611.329,E2 -24611.329} C_VEL
LIN {X 0,Y 174.552,Z 423.941,A -85,B 0,C 180,E1 -24614.799,E2 -24614.799} C_VEL
LIN {X 0,Y 182.264,Z 417.501,A -85,B 0,C 180,E1 -24617.109,E2 -24617.109} C_VEL
LIN {X 0,Y 190.437,Z 409.543,A -85,B 0,C 180,E1 -24619.162,E2 -24619.162} C_VEL
LIN {X 0,Y 197.607,Z 401.557,A -85,B 0,C 180,E1 -24620.675,E2 -24620.675} C_VEL
LIN {X 0,Y 205.805,Z 390.801,A -85,B 0,C 180,E1 -24622.157,E2 -24622.157} C_VEL
LIN {X 0,Y 212.041,Z 380.976,A -85,B 0,C 180,E1 -24623.164,E2 -24623.164} C_VEL
LIN {X 0,Y 218.203,Z 369.165,A -85,B 0,C 180,E1 -24624.044,E2 -24624.044} C_VEL
LIN {X 0,Y 223.246,Z 357.179,A -85,B 0,C 180,E1 -24624.708,E2 -24624.708} C_VEL
LIN {X 0,Y 227.503,Z 343.519,A -85,B 0,C 180,E1 -24625.316,E2 -24625.316} C_VEL
LIN {X 0,Y 227.494,Z 342.684,A -85,B 0,C 180,E1 -24626.525,E2 -24626.525} C_VEL
LIN {X 0,Y 227.515,Z 342.653,A -85,B 0,C 180,E1 -24628.516,E2 -24628.516} C_VEL
LIN {X 0,Y 223.457,Z 355.381,A -85,B 0,C 180,E1 -24629.314,E2 -24629.314} C_VEL
LIN {X 0,Y 217.988,Z 367.95,A -85,B 0,C 180,E1 -24630.374,E2 -24630.374} C_VEL
LIN {X 0,Y 212.053,Z 378.62,A -85,B 0,C 180,E1 -24631.547,E2 -24631.547} C_VEL
LIN {X 0,Y 206.117,Z 387.516,A -85,B 0,C 180,E1 -24632.826,E2 -24632.826} C_VEL
LIN {X 0,Y 199.335,Z 395.941,A -85,B 0,C 180,E1 -24634.411,E2 -24634.411} C_VEL
LIN {X 0,Y 190.818,Z 404.701,A -85,B 0,C 180,E1 -24636.617,E2 -24636.617} C_VEL
LIN {X 0,Y 183.77,Z 410.697,A -85,B 0,C 180,E1 -24638.695,E2 -24638.695} C_VEL
LIN {X 0,Y 175.85,Z 416.209,A -85,B 0,C 180,E1 -24641.352,E2 -24641.352} C_VEL
LIN {X 0,Y 167.629,Z 420.677,A -85,B 0,C 180,E1 -24644.647,E2 -24644.647} C_VEL
LIN {X 0,Y 161.683,Z 423.052,A -85,B 0,C 180,E1 -24647.446,E2 -24647.446} C_VEL
LIN {X 0,Y 157.001,Z 424.359,A -85,B 0,C 180,E1 -24650.007,E2 -24650.007} C_VEL
LIN {X 0,Y 153.601,Z 424.92,A -85,B 0,C 180,E1 -24652.109,E2 -24652.109} C_VEL
LIN {X 0,Y 147.91,Z 424.986,A -85,B 0,C 180,E1 -24656.239,E2 -24656.239} C_VEL
LIN {X 0,Y 143.811,Z 424.002,A -85,B 0,C 180,E1 -24659.999,E2 -24659.999} C_VEL
LIN {X 0,Y 140.823,Z 422.337,A -85,B 0,C 180,E1 -24663.478,E2 -24663.478} C_VEL
LIN {X 0,Y 138.267,Z 419.755,A -85,B 0,C 180,E1 -24667.299,E2 -24667.299} C_VEL
LIN {X 0,Y 136.132,Z 415.616,A -85,B 0,C 180,E1 -24671.916,E2 -24671.916} C_VEL
LIN {X 0,Y 134.829,Z 410.078,A -85,B 0,C 180,E1 -24676.658,E2 -24676.658} C_VEL
LIN {X 0,Y 134.451,Z 402.909,A -85,B 0,C 180,E1 -24681.462,E2 -24681.462} C_VEL
LIN {X 0,Y 134.807,Z 395.424,A -85,B 0,C 180,E1 -24685.473,E2 -24685.473} C_VEL
LIN {X 0,Y 135.423,Z 386.003,A -85,B 0,C 180,E1 -24689.537,E2 -24689.537} C_VEL
LIN {X 0,Y 136.437,Z 375.298,A -85,B 0,C 180,E1 -24693.18,E2 -24693.18} C_VEL
LIN {X 0,Y 137.639,Z 363.294,A -85,B 0,C 180,E1 -24696.334,E2 -24696.334} C_VEL
LIN {X 0,Y 138.821,Z 351.045,A -85,B 0,C 180,E1 -24698.791,E2 -24698.791} C_VEL
LIN {X 0,Y 139.825,Z 338.304,A -85,B 0,C 180,E1 -24700.679,E2 -24700.679} C_VEL
LIN {X 0,Y 140.612,Z 324.506,A -85,B 0,C 180,E1 -24702.069,E2 -24702.069} C_VEL
LIN {X 0,Y 143.42,Z 268.852,A -85,B 0,C 180,E1 -24706.439,E2 -24706.439} C_VEL
LIN {X 0,Y 141.355,Z 250.178,A -85,B 0,C 180,E1 -24708.078,E2 -24708.078} C_VEL
LIN {X 0,Y 138.632,Z 239.528,A -85,B 0,C 180,E1 -24709.257,E2 -24709.257} C_VEL
LIN {X 0,Y 136.735,Z 230.036,A -85,B 0,C 180,E1 -24714.672,E2 -24714.672} C_VEL
LIN {X 0,Y 136.21,Z 227.671,A -85,B 0,C 180,E1 -24716.237,E2 -24716.237} C_VEL
LIN {X 0,Y 136.148,Z 227.525,A -85,B 0,C 180,E1 -24722.315,E2 -24722.315} C_VEL
LIN {X 0,Y 136.243,Z 227.513,A -85,B 0,C 180,E1 -24728.831,E2 -24728.831} C_VEL
LIN {X 0,Y 136.276,Z 227.508,A -85,B 0,C 180,E1 -24735.055,E2 -24735.055} C_VEL
LIN {X 0,Y 136.499,Z 227.481,A -85,B 0,C 180,E1 -24738.113,E2 -24738.113} C_VEL
LIN {X 0,Y 136.605,Z 227.463,A -85,B 0,C 180,E1 -24741.119,E2 -24741.119} C_VEL
LIN {X 0,Y 137.132,Z 227.397,A -85,B 0,C 180,E1 -24749.998,E2 -24749.998} C_VEL
LIN {X 0,Y 136.589,Z 227.465,A -85,B 0,C 180,E1 -24758.878,E2 -24758.878} C_VEL
LIN {X 0,Y 136.487,Z 227.483,A -85,B 0,C 180,E1 -24761.952,E2 -24761.952} C_VEL
LIN {X 0,Y 136.24,Z 227.51,A -85,B 0,C 180,E1 -24768.027,E2 -24768.027} C_VEL
LIN {X 0,Y 136.194,Z 227.519,A -85,B 0,C 180,E1 -24771.747,E2 -24771.747} C_VEL
LIN {X 0,Y 136.111,Z 227.531,A -85,B 0,C 180,E1 -24778.627,E2 -24778.627} C_VEL
LIN {X 0,Y 136.077,Z 227.531,A -85,B 0,C 180,E1 -24784.616,E2 -24784.616} C_VEL
LIN {X 0,Y 136.084,Z 227.532,A -85,B 0,C 180,E1 -24789.227,E2 -24789.227} C_VEL
LIN {X 0,Y 136.09,Z 227.53,A -85,B 0,C 180,E1 -24793.7,E2 -24793.7} C_VEL
LIN {X 0,Y 136.091,Z 227.532,A -85,B 0,C 180,E1 -24797.831,E2 -24797.831} C_VEL
LIN {X 0,Y 136.072,Z 227.531,A -85,B 0,C 180,E1 -24801.701,E2 -24801.701} C_VEL
LIN {X 0,Y 136.085,Z 227.533,A -85,B 0,C 180,E1 -24805.717,E2 -24805.717} C_VEL
LIN {X 0,Y 136.14,Z 227.527,A -85,B 0,C 180,E1 -24812.317,E2 -24812.317} C_VEL
LIN {X 0,Y 136.237,Z 227.512,A -85,B 0,C 180,E1 -24818.833,E2 -24818.833} C_VEL
LIN {X 0,Y 136.258,Z 227.506,A -85,B 0,C 180,E1 -24825.056,E2 -24825.056} C_VEL
LIN {X 0,Y 136.425,Z 227.492,A -85,B 0,C 180,E1 -24828.166,E2 -24828.166} C_VEL
LIN {X 0,Y 136.545,Z 227.475,A -85,B 0,C 180,E1 -24831.119,E2 -24831.119} C_VEL
LIN {X 0,Y 137.127,Z 227.401,A -85,B 0,C 180,E1 -24840.001,E2 -24840.001} C_VEL
LIN {X 0,Y 136.586,Z 227.469,A -85,B 0,C 180,E1 -24848.881,E2 -24848.881} C_VEL
LIN {X 0,Y 136.487,Z 227.482,A -85,B 0,C 180,E1 -24851.956,E2 -24851.956} C_VEL
LIN {X 0,Y 136.238,Z 227.509,A -85,B 0,C 180,E1 -24858.032,E2 -24858.032} C_VEL
LIN {X 0,Y 136.194,Z 227.52,A -85,B 0,C 180,E1 -24861.751,E2 -24861.751} C_VEL
LIN {X 0,Y 136.097,Z 227.529,A -85,B 0,C 180,E1 -24868.618,E2 -24868.618} C_VEL
LIN {X 0,Y 136.04,Z 227.54,A -85,B 0,C 180,E1 -24874.632,E2 -24874.632} C_VEL
LIN {X 0,Y 136.025,Z 227.541,A -85,B 0,C 180,E1 -24879.199,E2 -24879.199} C_VEL
LIN {X 0,Y 136.079,Z 227.782,A -85,B 0,C 180,E1 -24884.655,E2 -24884.655} C_VEL
LIN {X 0,Y 138.485,Z 238.274,A -85,B 0,C 180,E1 -24890.484,E2 -24890.484} C_VEL
LIN {X 0,Y 141.324,Z 250.995,A -85,B 0,C 180,E1 -24897.015,E2 -24897.015} C_VEL
LIN {X 0,Y 141.61,Z 252.401,A -85,B 0,C 180,E1 -24897.535,E2 -24897.535} C_VEL
LIN {X 0,Y 141.721,Z 256.401,A -85,B 0,C 180,E1 -24897.887,E2 -24897.887} C_VEL
LIN {X 0,Y 142.029,Z 278.407,A -85,B 0,C 180,E1 -24899.577,E2 -24899.577} C_VEL
LIN {X 0,Y 143.382,Z 306.351,A -85,B 0,C 180,E1 -24901.737,E2 -24901.737} C_VEL
LIN {X 0,Y 141.367,Z 352.374,A -85,B 0,C 180,E1 -24905.202,E2 -24905.202} C_VEL
LIN {X 0,Y 140.612,Z 364.459,A -85,B 0,C 180,E1 -24906.629,E2 -24906.629} C_VEL
LIN {X 0,Y 139.48,Z 376.241,A -85,B 0,C 180,E1 -24908.576,E2 -24908.576} C_VEL
LIN {X 0,Y 138.296,Z 387.75,A -85,B 0,C 180,E1 -24911.099,E2 -24911.099} C_VEL
LIN {X 0,Y 137.213,Z 398.109,A -85,B 0,C 180,E1 -24914.022,E2 -24914.022} C_VEL
LIN {X 0,Y 136.434,Z 407.534,A -85,B 0,C 180,E1 -24917.356,E2 -24917.356} C_VEL
LIN {X 0,Y 136.107,Z 416.078,A -85,B 0,C 180,E1 -24921.091,E2 -24921.091} C_VEL
LIN {X 0,Y 136.303,Z 424.155,A -85,B 0,C 180,E1 -24925.566,E2 -24925.566} C_VEL
LIN {X 0,Y 136.673,Z 430.311,A -85,B 0,C 180,E1 -24930.002,E2 -24930.002} C_VEL
LIN {X 0,Y 136.642,Z 431.921,A -85,B 0,C 180,E1 -24931.476,E2 -24931.476} C_VEL
LIN {X 0,Y 135.596,Z 435.642,A -85,B 0,C 180,E1 -24935.952,E2 -24935.952} C_VEL
LIN {X 0,Y 135.155,Z 437.551,A -85,B 0,C 180,E1 -24938.977,E2 -24938.977} C_VEL
LIN {X 0,Y 135.601,Z 440.147,A -85,B 0,C 180,E1 -24945.021,E2 -24945.021} C_VEL
LIN {X 0,Y 137.847,Z 441.352,A -85,B 0,C 180,E1 -24950.911,E2 -24950.911} C_VEL
LIN {X 0,Y 141.894,Z 441.195,A -85,B 0,C 180,E1 -24956.474,E2 -24956.474} C_VEL
LIN {X 0,Y 147.413,Z 439.611,A -85,B 0,C 180,E1 -24961.632,E2 -24961.632} C_VEL
LIN {X 0,Y 151.825,Z 437.782,A -85,B 0,C 180,E1 -24964.742,E2 -24964.742} C_VEL
LIN {X 0,Y 154.347,Z 436.427,A -85,B 0,C 180,E1 -24966.674,E2 -24966.674} C_VEL
LIN {X 0,Y 158.69,Z 432.694,A -85,B 0,C 180,E1 -24971.306,E2 -24971.306} C_VEL
LIN {X 0,Y 161.998,Z 430.115,A -85,B 0,C 180,E1 -24973.685,E2 -24973.685} C_VEL
LIN {X 0,Y 164.267,Z 428.617,A -85,B 0,C 180,E1 -24974.681,E2 -24974.681} C_VEL
LIN {X 0,Y 173.529,Z 422.257,A -85,B 0,C 180,E1 -24977.659,E2 -24977.659} C_VEL
LIN {X 0,Y 183.134,Z 414.42,A -85,B 0,C 180,E1 -24980.134,E2 -24980.134} C_VEL
LIN {X 0,Y 191.792,Z 406.048,A -85,B 0,C 180,E1 -24981.986,E2 -24981.986} C_VEL
LIN {X 0,Y 199.372,Z 397.442,A -85,B 0,C 180,E1 -24983.319,E2 -24983.319} C_VEL
LIN {X 0,Y 207.083,Z 387.114,A -85,B 0,C 180,E1 -24984.541,E2 -24984.541} C_VEL
LIN {X 0,Y 214.168,Z 375.626,A -85,B 0,C 180,E1 -24985.512,E2 -24985.512} C_VEL
LIN {X 0,Y 220.357,Z 363.049,A -85,B 0,C 180,E1 -24986.275,E2 -24986.275} C_VEL
LIN {X 0,Y 224.52,Z 352.295,A -85,B 0,C 180,E1 -24986.74,E2 -24986.74} C_VEL
LIN {X 0,Y 224.902,Z 351.026,A -85,B 0,C 180,E1 -24987.167,E2 -24987.167} C_VEL
LIN {X 0,Y 219.689,Z 364.035,A -85,B 0,C 180,E1 -24988.09,E2 -24988.09} C_VEL
LIN {X 0,Y 213.424,Z 375.915,A -85,B 0,C 180,E1 -24989.198,E2 -24989.198} C_VEL
LIN {X 0,Y 206.757,Z 385.984,A -85,B 0,C 180,E1 -24990.469,E2 -24990.469} C_VEL
LIN {X 0,Y 198.692,Z 395.947,A -85,B 0,C 180,E1 -24992.166,E2 -24992.166} C_VEL
LIN {X 0,Y 190.333,Z 404.372,A -85,B 0,C 180,E1 -24994.125,E2 -24994.125} C_VEL
LIN {X 0,Y 182.645,Z 410.751,A -85,B 0,C 180,E1 -24996.169,E2 -24996.169} C_VEL
LIN {X 0,Y 173.041,Z 417.183,A -85,B 0,C 180,E1 -24999.092,E2 -24999.092} C_VEL
LIN {X 0,Y 166.258,Z 420.733,A -85,B 0,C 180,E1 -25001.515,E2 -25001.515} C_VEL
LIN {X 0,Y 158.949,Z 423.629,A -85,B 0,C 180,E1 -25004.614,E2 -25004.614} C_VEL
LIN {X 0,Y 153.181,Z 425.135,A -85,B 0,C 180,E1 -25007.468,E2 -25007.468} C_VEL
LIN {X 0,Y 150.09,Z 425.707,A -85,B 0,C 180,E1 -25009.203,E2 -25009.203} C_VEL
LIN {X 0,Y 146.1,Z 425.97,A -85,B 0,C 180,E1 -25011.701,E2 -25011.701} C_VEL
LIN {X 0,Y 141.003,Z 425.531,A -85,B 0,C 180,E1 -25015.475,E2 -25015.475} C_VEL
LIN {X 0,Y 136.233,Z 423.879,A -85,B 0,C 180,E1 -25019.999,E2 -25019.999} C_VEL
LIN {X 0,Y 132.649,Z 421.152,A -85,B 0,C 180,E1 -25024.555,E2 -25024.555} C_VEL
LIN {X 0,Y 129.983,Z 417.198,A -85,B 0,C 180,E1 -25029.333,E2 -25029.333} C_VEL
LIN {X 0,Y 128.233,Z 411.933,A -85,B 0,C 180,E1 -25034.277,E2 -25034.277} C_VEL
LIN {X 0,Y 127.471,Z 405.156,A -85,B 0,C 180,E1 -25039.316,E2 -25039.316} C_VEL
LIN {X 0,Y 127.565,Z 398.102,A -85,B 0,C 180,E1 -25043.541,E2 -25043.541} C_VEL
LIN {X 0,Y 128.063,Z 389.76,A -85,B 0,C 180,E1 -25047.587,E2 -25047.587} C_VEL
LIN {X 0,Y 128.959,Z 379.326,A -85,B 0,C 180,E1 -25051.636,E2 -25051.636} C_VEL
LIN {X 0,Y 130.062,Z 367.712,A -85,B 0,C 180,E1 -25055.157,E2 -25055.157} C_VEL
LIN {X 0,Y 131.264,Z 355.526,A -85,B 0,C 180,E1 -25058.002,E2 -25058.002} C_VEL
LIN {X 0,Y 132.316,Z 343.699,A -85,B 0,C 180,E1 -25060.091,E2 -25060.091} C_VEL
LIN {X 0,Y 133.216,Z 330.261,A -85,B 0,C 180,E1 -25061.761,E2 -25061.761} C_VEL
LIN {X 0,Y 136.353,Z 268.749,A -85,B 0,C 180,E1 -25066.893,E2 -25066.893} C_VEL
LIN {X 0,Y 134.457,Z 251.551,A -85,B 0,C 180,E1 -25068.479,E2 -25068.479} C_VEL
LIN {X 0,Y 131.513,Z 240.028,A -85,B 0,C 180,E1 -25069.785,E2 -25069.785} C_VEL
LIN {X 0,Y 129.824,Z 231.654,A -85,B 0,C 180,E1 -25074.738,E2 -25074.738} C_VEL
LIN {X 0,Y 129.189,Z 228.742,A -85,B 0,C 180,E1 -25076.64,E2 -25076.64} C_VEL
LIN {X 0,Y 129.069,Z 228.408,A -85,B 0,C 180,E1 -25077.932,E2 -25077.932} C_VEL
LIN {X 0,Y 129.031,Z 228.411,A -85,B 0,C 180,E1 -25084.165,E2 -25084.165} C_VEL
LIN {X 0,Y 129.107,Z 228.401,A -85,B 0,C 180,E1 -25087.725,E2 -25087.725} C_VEL
LIN {X 0,Y 129.154,Z 228.398,A -85,B 0,C 180,E1 -25090.942,E2 -25090.942} C_VEL
LIN {X 0,Y 129.417,Z 228.364,A -85,B 0,C 180,E1 -25097.814,E2 -25097.814} C_VEL
LIN {X 0,Y 129.528,Z 228.346,A -85,B 0,C 180,E1 -25100.63,E2 -25100.63} C_VEL
LIN {X 0,Y 130.087,Z 228.274,A -85,B 0,C 180,E1 -25109.998,E2 -25109.998} C_VEL
LIN {X 0,Y 129.514,Z 228.349,A -85,B 0,C 180,E1 -25119.367,E2 -25119.367} C_VEL
LIN {X 0,Y 129.389,Z 228.368,A -85,B 0,C 180,E1 -25122.546,E2 -25122.546} C_VEL
LIN {X 0,Y 129.151,Z 228.397,A -85,B 0,C 180,E1 -25129.054,E2 -25129.054} C_VEL
LIN {X 0,Y 129.104,Z 228.403,A -85,B 0,C 180,E1 -25132.397,E2 -25132.397} C_VEL
LIN {X 0,Y 129.031,Z 228.412,A -85,B 0,C 180,E1 -25139.372,E2 -25139.372} C_VEL
LIN {X 0,Y 129.019,Z 228.412,A -85,B 0,C 180,E1 -25145.208,E2 -25145.208} C_VEL
LIN {X 0,Y 129.008,Z 228.409,A -85,B 0,C 180,E1 -25150.82,E2 -25150.82} C_VEL
LIN {X 0,Y 129.018,Z 228.413,A -85,B 0,C 180,E1 -25155.081,E2 -25155.081} C_VEL
LIN {X 0,Y 129,Z 228.411,A -85,B 0,C 180,E1 -25159.701,E2 -25159.701} C_VEL
LIN {X 0,Y 129.016,Z 228.414,A -85,B 0,C 180,E1 -25164.792,E2 -25164.792} C_VEL
LIN {X 0,Y 129.027,Z 228.412,A -85,B 0,C 180,E1 -25170.647,E2 -25170.647} C_VEL
LIN {X 0,Y 129.102,Z 228.397,A -85,B 0,C 180,E1 -25177.602,E2 -25177.602} C_VEL
LIN {X 0,Y 129.145,Z 228.397,A -85,B 0,C 180,E1 -25180.944,E2 -25180.944} C_VEL
LIN {X 0,Y 129.37,Z 228.369,A -85,B 0,C 180,E1 -25187.904,E2 -25187.904} C_VEL
LIN {X 0,Y 129.468,Z 228.357,A -85,B 0,C 180,E1 -25190.629,E2 -25190.629} C_VEL
LIN {X 0,Y 130.083,Z 228.279,A -85,B 0,C 180,E1 -25200.001,E2 -25200.001} C_VEL
LIN {X 0,Y 129.512,Z 228.348,A -85,B 0,C 180,E1 -25209.371,E2 -25209.371} C_VEL
LIN {X 0,Y 129.388,Z 228.365,A -85,B 0,C 180,E1 -25212.55,E2 -25212.55} C_VEL
LIN {X 0,Y 129.149,Z 228.391,A -85,B 0,C 180,E1 -25219.058,E2 -25219.058} C_VEL
LIN {X 0,Y 129.105,Z 228.402,A -85,B 0,C 180,E1 -25222.401,E2 -25222.401} C_VEL
LIN {X 0,Y 129.026,Z 228.409,A -85,B 0,C 180,E1 -25225.835,E2 -25225.835} C_VEL
LIN {X 0,Y 129.013,Z 228.414,A -85,B 0,C 180,E1 -25229.36,E2 -25229.36} C_VEL
LIN {X 0,Y 128.956,Z 228.422,A -85,B 0,C 180,E1 -25235.17,E2 -25235.17} C_VEL
LIN {X 0,Y 128.928,Z 228.425,A -85,B 0,C 180,E1 -25240.856,E2 -25240.856} C_VEL
LIN {X 0,Y 129.028,Z 228.633,A -85,B 0,C 180,E1 -25243.987,E2 -25243.987} C_VEL
LIN {X 0,Y 131.387,Z 239.033,A -85,B 0,C 180,E1 -25250.07,E2 -25250.07} C_VEL
LIN {X 0,Y 134.068,Z 250.986,A -85,B 0,C 180,E1 -25256.558,E2 -25256.558} C_VEL
LIN {X 0,Y 134.366,Z 252.392,A -85,B 0,C 180,E1 -25257.01,E2 -25257.01} C_VEL
LIN {X 0,Y 134.786,Z 255.322,A -85,B 0,C 180,E1 -25257.306,E2 -25257.306} C_VEL
LIN {X 0,Y 134.902,Z 276.546,A -85,B 0,C 180,E1 -25259.011,E2 -25259.011} C_VEL
LIN {X 0,Y 136.342,Z 306.22,A -85,B 0,C 180,E1 -25261.432,E2 -25261.432} C_VEL
LIN {X 0,Y 134.317,Z 351.699,A -85,B 0,C 180,E1 -25265.05,E2 -25265.05} C_VEL
LIN {X 0,Y 133.549,Z 363.778,A -85,B 0,C 180,E1 -25266.551,E2 -25266.551} C_VEL
LIN {X 0,Y 132.42,Z 375.585,A -85,B 0,C 180,E1 -25268.602,E2 -25268.602} C_VEL
LIN {X 0,Y 131.241,Z 387.089,A -85,B 0,C 180,E1 -25271.261,E2 -25271.261} C_VEL
LIN {X 0,Y 130.18,Z 397.385,A -85,B 0,C 180,E1 -25274.342,E2 -25274.342} C_VEL
LIN {X 0,Y 129.453,Z 407.402,A -85,B 0,C 180,E1 -25278.124,E2 -25278.124} C_VEL
LIN {X 0,Y 129.229,Z 415.998,A -85,B 0,C 180,E1 -25282.188,E2 -25282.188} C_VEL
LIN {X 0,Y 129.483,Z 422.712,A -85,B 0,C 180,E1 -25286.112,E2 -25286.112} C_VEL
LIN {X 0,Y 129.797,Z 428.042,A -85,B 0,C 180,E1 -25290.002,E2 -25290.002} C_VEL
LIN {X 0,Y 129.824,Z 429.826,A -85,B 0,C 180,E1 -25291.553,E2 -25291.553} C_VEL
LIN {X 0,Y 129.087,Z 432.61,A -85,B 0,C 180,E1 -25294.686,E2 -25294.686} C_VEL
LIN {X 0,Y 128.312,Z 435.915,A -85,B 0,C 180,E1 -25299.621,E2 -25299.621} C_VEL
LIN {X 0,Y 128.839,Z 438.748,A -85,B 0,C 180,E1 -25305.83,E2 -25305.83} C_VEL
LIN {X 0,Y 131.262,Z 440.279,A -85,B 0,C 180,E1 -25312.014,E2 -25312.014} C_VEL
LIN {X 0,Y 135.576,Z 440.433,A -85,B 0,C 180,E1 -25317.812,E2 -25317.812} C_VEL
LIN {X 0,Y 141.404,Z 439.244,A -85,B 0,C 180,E1 -25323.144,E2 -25323.144} C_VEL
LIN {X 0,Y 145.808,Z 437.765,A -85,B 0,C 180,E1 -25326.184,E2 -25326.184} C_VEL
LIN {X 0,Y 152.925,Z 434.791,A -85,B 0,C 180,E1 -25330.048,E2 -25330.048} C_VEL
LIN {X 0,Y 159.728,Z 431.278,A -85,B 0,C 180,E1 -25333.002,E2 -25333.002} C_VEL
LIN {X 0,Y 164.267,Z 428.617,A -85,B 0,C 180,E1 -25334.681,E2 -25334.681} C_VEL
LIN {X 0,Y 167.657,Z 426.308,A -85,B 0,C 180,E1 -25336.156,E2 -25336.156} C_VEL
LIN {X 0,Y 172.251,Z 422.368,A -85,B 0,C 180,E1 -25338.813,E2 -25338.813} C_VEL
LIN {X 0,Y 177.081,Z 417.869,A -85,B 0,C 180,E1 -25341.214,E2 -25341.214} C_VEL
LIN {X 0,Y 180.717,Z 414.697,A -85,B 0,C 180,E1 -25342.283,E2 -25342.283} C_VEL
LIN {X 0,Y 189.107,Z 407.119,A -85,B 0,C 180,E1 -25343.934,E2 -25343.934} C_VEL
LIN {X 0,Y 197.353,Z 398.498,A -85,B 0,C 180,E1 -25345.264,E2 -25345.264} C_VEL
LIN {X 0,Y 205.559,Z 388.146,A -85,B 0,C 180,E1 -25346.448,E2 -25346.448} C_VEL
LIN {X 0,Y 211.229,Z 379.67,A -85,B 0,C 180,E1 -25347.154,E2 -25347.154} C_VEL
LIN {X 0,Y 211.82,Z 378.631,A -85,B 0,C 180,E1 -25347.47,E2 -25347.47} C_VEL
LIN {X 0,Y 205.033,Z 388.251,A -85,B 0,C 180,E1 -25348.661,E2 -25348.661} C_VEL
LIN {X 0,Y 197.455,Z 397.111,A -85,B 0,C 180,E1 -25350.111,E2 -25350.111} C_VEL
LIN {X 0,Y 188.014,Z 406.048,A -85,B 0,C 180,E1 -25352.143,E2 -25352.143} C_VEL
LIN {X 0,Y 178.897,Z 413.044,A -85,B 0,C 180,E1 -25354.396,E2 -25354.396} C_VEL
LIN {X 0,Y 170.128,Z 418.404,A -85,B 0,C 180,E1 -25356.892,E2 -25356.892} C_VEL
LIN {X 0,Y 161.818,Z 422.337,A -85,B 0,C 180,E1 -25359.667,E2 -25359.667} C_VEL
LIN {X 0,Y 154.773,Z 424.797,A -85,B 0,C 180,E1 -25362.477,E2 -25362.477} C_VEL
LIN {X 0,Y 147.048,Z 426.454,A -85,B 0,C 180,E1 -25366.173,E2 -25366.173} C_VEL
LIN {X 0,Y 142.646,Z 426.83,A -85,B 0,C 180,E1 -25368.633,E2 -25368.633} C_VEL
LIN {X 0,Y 138.604,Z 426.709,A -85,B 0,C 180,E1 -25371.249,E2 -25371.249} C_VEL
LIN {X 0,Y 134.125,Z 425.907,A -85,B 0,C 180,E1 -25374.626,E2 -25374.626} C_VEL
LIN {X 0,Y 128.657,Z 423.436,A -85,B 0,C 180,E1 -25379.998,E2 -25379.998} C_VEL
LIN {X 0,Y 125.099,Z 420.083,A -85,B 0,C 180,E1 -25384.832,E2 -25384.832} C_VEL
LIN {X 0,Y 122.525,Z 415.535,A -85,B 0,C 180,E1 -25389.907,E2 -25389.907} C_VEL
LIN {X 0,Y 120.954,Z 409.575,A -85,B 0,C 180,E1 -25395.156,E2 -25395.156} C_VEL
LIN {X 0,Y 120.434,Z 401.971,A -85,B 0,C 180,E1 -25400.494,E2 -25400.494} C_VEL
LIN {X 0,Y 120.716,Z 394.125,A -85,B 0,C 180,E1 -25404.965,E2 -25404.965} C_VEL
LIN {X 0,Y 121.249,Z 386.065,A -85,B 0,C 180,E1 -25408.695,E2 -25408.695} C_VEL
LIN {X 0,Y 122.145,Z 375.464,A -85,B 0,C 180,E1 -25412.642,E2 -25412.642} C_VEL
LIN {X 0,Y 123.307,Z 364.076,A -85,B 0,C 180,E1 -25415.967,E2 -25415.967} C_VEL
LIN {X 0,Y 124.487,Z 352.171,A -85,B 0,C 180,E1 -25418.646,E2 -25418.646} C_VEL
LIN {X 0,Y 125.511,Z 339.677,A -85,B 0,C 180,E1 -25420.743,E2 -25420.743} C_VEL
LIN {X 0,Y 126.369,Z 326.347,A -85,B 0,C 180,E1 -25422.282,E2 -25422.282} C_VEL
LIN {X 0,Y 129.323,Z 269.171,A -85,B 0,C 180,E1 -25427.337,E2 -25427.337} C_VEL
LIN {X 0,Y 127.438,Z 252.513,A -85,B 0,C 180,E1 -25428.956,E2 -25428.956} C_VEL
LIN {X 0,Y 124.348,Z 240.36,A -85,B 0,C 180,E1 -25430.384,E2 -25430.384} C_VEL
LIN {X 0,Y 122.529,Z 231.425,A -85,B 0,C 180,E1 -25435.994,E2 -25435.994} C_VEL
LIN {X 0,Y 122.07,Z 229.38,A -85,B 0,C 180,E1 -25437.575,E2 -25437.575} C_VEL
LIN {X 0,Y 121.957,Z 229.293,A -85,B 0,C 180,E1 -25442.545,E2 -25442.545} C_VEL
LIN {X 0,Y 122.023,Z 229.284,A -85,B 0,C 180,E1 -25447.147,E2 -25447.147} C_VEL
LIN {X 0,Y 122.111,Z 229.269,A -85,B 0,C 180,E1 -25453.273,E2 -25453.273} C_VEL
LIN {X 0,Y 122.363,Z 229.243,A -85,B 0,C 180,E1 -25457.52,E2 -25457.52} C_VEL
LIN {X 0,Y 122.454,Z 229.227,A -85,B 0,C 180,E1 -25460.083,E2 -25460.083} C_VEL
LIN {X 0,Y 122.608,Z 229.212,A -85,B 0,C 180,E1 -25466.712,E2 -25466.712} C_VEL
LIN {X 0,Y 123.041,Z 229.152,A -85,B 0,C 180,E1 -25469.998,E2 -25469.998} C_VEL
LIN {X 0,Y 122.444,Z 229.23,A -85,B 0,C 180,E1 -25476.589,E2 -25476.589} C_VEL
LIN {X 0,Y 122.443,Z 229.23,A -85,B 0,C 180,E1 -25479.913,E2 -25479.913} C_VEL
LIN {X 0,Y 122.258,Z 229.255,A -85,B 0,C 180,E1 -25483.291,E2 -25483.291} C_VEL
LIN {X 0,Y 122.042,Z 229.282,A -85,B 0,C 180,E1 -25490.211,E2 -25490.211} C_VEL
LIN {X 0,Y 121.979,Z 229.286,A -85,B 0,C 180,E1 -25493.783,E2 -25493.783} C_VEL
LIN {X 0,Y 121.937,Z 229.296,A -85,B 0,C 180,E1 -25500.172,E2 -25500.172} C_VEL
LIN {X 0,Y 121.932,Z 229.295,A -85,B 0,C 180,E1 -25506.205,E2 -25506.205} C_VEL
LIN {X 0,Y 121.936,Z 229.289,A -85,B 0,C 180,E1 -25511.475,E2 -25511.475} C_VEL
LIN {X 0,Y 121.931,Z 229.293,A -85,B 0,C 180,E1 -25518.526,E2 -25518.526} C_VEL
LIN {X 0,Y 121.968,Z 229.292,A -85,B 0,C 180,E1 -25524.817,E2 -25524.817} C_VEL
LIN {X 0,Y 121.936,Z 229.291,A -85,B 0,C 180,E1 -25529.826,E2 -25529.826} C_VEL
LIN {X 0,Y 121.977,Z 229.285,A -85,B 0,C 180,E1 -25536.216,E2 -25536.216} C_VEL
LIN {X 0,Y 122.038,Z 229.282,A -85,B 0,C 180,E1 -25539.787,E2 -25539.787} C_VEL
LIN {X 0,Y 122.232,Z 229.256,A -85,B 0,C 180,E1 -25546.705,E2 -25546.705} C_VEL
LIN {X 0,Y 122.401,Z 229.238,A -85,B 0,C 180,E1 -25550.083,E2 -25550.083} C_VEL
LIN {X 0,Y 122.592,Z 229.213,A -85,B 0,C 180,E1 -25556.715,E2 -25556.715} C_VEL
LIN {X 0,Y 123.036,Z 229.156,A -85,B 0,C 180,E1 -25560.002,E2 -25560.002} C_VEL
LIN {X 0,Y 122.442,Z 229.232,A -85,B 0,C 180,E1 -25566.594,E2 -25566.594} C_VEL
LIN {X 0,Y 122.441,Z 229.226,A -85,B 0,C 180,E1 -25569.917,E2 -25569.917} C_VEL
LIN {X 0,Y 122.257,Z 229.255,A -85,B 0,C 180,E1 -25573.295,E2 -25573.295} C_VEL
LIN {X 0,Y 122.041,Z 229.279,A -85,B 0,C 180,E1 -25580.215,E2 -25580.215} C_VEL
LIN {X 0,Y 121.98,Z 229.29,A -85,B 0,C 180,E1 -25583.787,E2 -25583.787} C_VEL
LIN {X 0,Y 121.923,Z 229.297,A -85,B 0,C 180,E1 -25590.164,E2 -25590.164} C_VEL
LIN {X 0,Y 121.88,Z 229.301,A -85,B 0,C 180,E1 -25596.173,E2 -25596.173} C_VEL
LIN {X 0,Y 121.942,Z 229.461,A -85,B 0,C 180,E1 -25603.262,E2 -25603.262} C_VEL
LIN {X 0,Y 124.314,Z 239.938,A -85,B 0,C 180,E1 -25609.751,E2 -25609.751} C_VEL
LIN {X 0,Y 126.63,Z 250.199,A -85,B 0,C 180,E1 -25615.648,E2 -25615.648} C_VEL
LIN {X 0,Y 126.979,Z 251.736,A -85,B 0,C 180,E1 -25616.338,E2 -25616.338} C_VEL
LIN {X 0,Y 127.804,Z 255.701,A -85,B 0,C 180,E1 -25616.779,E2 -25616.779} C_VEL
LIN {X 0,Y 127.903,Z 277.072,A -85,B 0,C 180,E1 -25618.594,E2 -25618.594} C_VEL
LIN {X 0,Y 129.249,Z 306.659,A -85,B 0,C 180,E1 -25621.149,E2 -25621.149} C_VEL
LIN {X 0,Y 127.223,Z 351.499,A -85,B 0,C 180,E1 -25624.982,E2 -25624.982} C_VEL
LIN {X 0,Y 126.52,Z 362.754,A -85,B 0,C 180,E1 -25626.471,E2 -25626.471} C_VEL
LIN {X 0,Y 125.39,Z 374.592,A -85,B 0,C 180,E1 -25628.637,E2 -25628.637} C_VEL
LIN {X 0,Y 124.225,Z 386.078,A -85,B 0,C 180,E1 -25631.447,E2 -25631.447} C_VEL
LIN {X 0,Y 123.209,Z 396.462,A -85,B 0,C 180,E1 -25634.706,E2 -25634.706} C_VEL
LIN {X 0,Y 122.517,Z 406.61,A -85,B 0,C 180,E1 -25638.747,E2 -25638.747} C_VEL
LIN {X 0,Y 122.365,Z 414.39,A -85,B 0,C 180,E1 -25642.577,E2 -25642.577} C_VEL
LIN {X 0,Y 122.694,Z 422.419,A -85,B 0,C 180,E1 -25647.54,E2 -25647.54} C_VEL
LIN {X 0,Y 122.966,Z 425.706,A -85,B 0,C 180,E1 -25650.002,E2 -25650.002} C_VEL
LIN {X 0,Y 123.039,Z 427.593,A -85,B 0,C 180,E1 -25651.639,E2 -25651.639} C_VEL
LIN {X 0,Y 122.306,Z 430.548,A -85,B 0,C 180,E1 -25654.947,E2 -25654.947} C_VEL
LIN {X 0,Y 121.498,Z 434.276,A -85,B 0,C 180,E1 -25660.459,E2 -25660.459} C_VEL
LIN {X 0,Y 122.126,Z 437.262,A -85,B 0,C 180,E1 -25666.725,E2 -25666.725} C_VEL
LIN {X 0,Y 124.754,Z 439.072,A -85,B 0,C 180,E1 -25673.227,E2 -25673.227} C_VEL
LIN {X 0,Y 129.342,Z 439.607,A -85,B 0,C 180,E1 -25679.279,E2 -25679.279} C_VEL
LIN {X 0,Y 135.517,Z 438.77,A -85,B 0,C 180,E1 -25684.785,E2 -25684.785} C_VEL
LIN {X 0,Y 143.198,Z 436.564,A -85,B 0,C 180,E1 -25689.647,E2 -25689.647} C_VEL
LIN {X 0,Y 152.214,Z 432.965,A -85,B 0,C 180,E1 -25693.837,E2 -25693.837} C_VEL
LIN {X 0,Y 162.248,Z 427.69,A -85,B 0,C 180,E1 -25697.426,E2 -25697.426} C_VEL
LIN {X 0,Y 170.251,Z 422.615,A -85,B 0,C 180,E1 -25699.792,E2 -25699.792} C_VEL
LIN {X 0,Y 180.19,Z 415.139,A -85,B 0,C 180,E1 -25702.17,E2 -25702.17} C_VEL
LIN {X 0,Y 180.717,Z 414.697,A -85,B 0,C 180,E1 -25702.283,E2 -25702.283} C_VEL
LIN {X 0,Y 183.126,Z 412.534,A -85,B 0,C 180,E1 -25703.028,E2 -25703.028} C_VEL
LIN {X 0,Y 189.321,Z 405.961,A -85,B 0,C 180,E1 -25706.122,E2 -25706.122} C_VEL
LIN {X 0,Y 191.729,Z 403.487,A -85,B 0,C 180,E1 -25706.708,E2 -25706.708} C_VEL
LIN {X 0,Y 196.315,Z 398.703,A -85,B 0,C 180,E1 -25707.353,E2 -25707.353} C_VEL
LIN {X 0,Y 197.852,Z 396.922,A -85,B 0,C 180,E1 -25707.803,E2 -25707.803} C_VEL
LIN {X 0,Y 189.858,Z 404.59,A -85,B 0,C 180,E1 -25709.334,E2 -25709.334} C_VEL
LIN {X 0,Y 181.594,Z 411.111,A -85,B 0,C 180,E1 -25711.067,E2 -25711.067} C_VEL
LIN {X 0,Y 172.26,Z 417.134,A -85,B 0,C 180,E1 -25713.333,E2 -25713.333} C_VEL
LIN {X 0,Y 163.496,Z 421.57,A -85,B 0,C 180,E1 -25715.789,E2 -25715.789} C_VEL
LIN {X 0,Y 154.812,Z 424.833,A -85,B 0,C 180,E1 -25718.703,E2 -25718.703} C_VEL
LIN {X 0,Y 148.467,Z 426.517,A -85,B 0,C 180,E1 -25721.221,E2 -25721.221} C_VEL
LIN {X 0,Y 139.669,Z 427.69,A -85,B 0,C 180,E1 -25725.427,E2 -25725.427} C_VEL
LIN {X 0,Y 135.195,Z 427.63,A -85,B 0,C 180,E1 -25727.997,E2 -25727.997} C_VEL
LIN {X 0,Y 131.061,Z 427.125,A -85,B 0,C 180,E1 -25730.741,E2 -25730.741} C_VEL
LIN {X 0,Y 127.278,Z 426.094,A -85,B 0,C 180,E1 -25733.694,E2 -25733.694} C_VEL
LIN {X 0,Y 123.968,Z 424.624,A -85,B 0,C 180,E1 -25736.748,E2 -25736.748} C_VEL
LIN {X 0,Y 119.554,Z 421.222,A -85,B 0,C 180,E1 -25742.022,E2 -25742.022} C_VEL
LIN {X 0,Y 116.62,Z 417.091,A -85,B 0,C 180,E1 -25746.921,E2 -25746.921} C_VEL
LIN {X 0,Y 114.454,Z 411.057,A -85,B 0,C 180,E1 -25752.712,E2 -25752.712} C_VEL
LIN {X 0,Y 113.527,Z 404.189,A -85,B 0,C 180,E1 -25758.029,E2 -25758.029} C_VEL
LIN {X 0,Y 113.538,Z 396.686,A -85,B 0,C 180,E1 -25762.758,E2 -25762.758} C_VEL
LIN {X 0,Y 113.997,Z 388.431,A -85,B 0,C 180,E1 -25767.042,E2 -25767.042} C_VEL
LIN {X 0,Y 114.843,Z 377.996,A -85,B 0,C 180,E1 -25771.387,E2 -25771.387} C_VEL
LIN {X 0,Y 115.768,Z 368.125,A -85,B 0,C 180,E1 -25774.688,E2 -25774.688} C_VEL
LIN {X 0,Y 117.029,Z 355.731,A -85,B 0,C 180,E1 -25777.878,E2 -25777.878} C_VEL
LIN {X 0,Y 118.084,Z 343.994,A -85,B 0,C 180,E1 -25780.145,E2 -25780.145} C_VEL
LIN {X 0,Y 118.999,Z 331.254,A -85,B 0,C 180,E1 -25781.919,E2 -25781.919} C_VEL
LIN {X 0,Y 122.23,Z 269.118,A -85,B 0,C 180,E1 -25787.79,E2 -25787.79} C_VEL
LIN {X 0,Y 120.596,Z 254.164,A -85,B 0,C 180,E1 -25789.33,E2 -25789.33} C_VEL
LIN {X 0,Y 117.188,Z 240.716,A -85,B 0,C 180,E1 -25791.018,E2 -25791.018} C_VEL
LIN {X 0,Y 115.705,Z 233.425,A -85,B 0,C 180,E1 -25795.814,E2 -25795.814} C_VEL
LIN {X 0,Y 115.016,Z 230.282,A -85,B 0,C 180,E1 -25798.232,E2 -25798.232} C_VEL
LIN {X 0,Y 114.946,Z 230.167,A -85,B 0,C 180,E1 -25806.505,E2 -25806.505} C_VEL
LIN {X 0,Y 115.013,Z 230.155,A -85,B 0,C 180,E1 -25812.208,E2 -25812.208} C_VEL
LIN {X 0,Y 115.285,Z 230.126,A -85,B 0,C 180,E1 -25817.255,E2 -25817.255} C_VEL
LIN {X 0,Y 115.391,Z 230.108,A -85,B 0,C 180,E1 -25819.469,E2 -25819.469} C_VEL
LIN {X 0,Y 115.534,Z 230.093,A -85,B 0,C 180,E1 -25826.51,E2 -25826.51} C_VEL
LIN {X 0,Y 115.993,Z 230.03,A -85,B 0,C 180,E1 -25829.998,E2 -25829.998} C_VEL
LIN {X 0,Y 115.386,Z 230.106,A -85,B 0,C 180,E1 -25836.994,E2 -25836.994} C_VEL
LIN {X 0,Y 115.281,Z 230.126,A -85,B 0,C 180,E1 -25842.736,E2 -25842.736} C_VEL
LIN {X 0,Y 115.01,Z 230.155,A -85,B 0,C 180,E1 -25847.788,E2 -25847.788} C_VEL
LIN {X 0,Y 114.942,Z 230.163,A -85,B 0,C 180,E1 -25853.49,E2 -25853.49} C_VEL
LIN {X 0,Y 114.864,Z 230.174,A -85,B 0,C 180,E1 -25861.067,E2 -25861.067} C_VEL
LIN {X 0,Y 114.843,Z 230.179,A -85,B 0,C 180,E1 -25867.728,E2 -25867.728} C_VEL
LIN {X 0,Y 114.859,Z 230.173,A -85,B 0,C 180,E1 -25872.758,E2 -25872.758} C_VEL
LIN {X 0,Y 114.859,Z 230.176,A -85,B 0,C 180,E1 -25877.698,E2 -25877.698} C_VEL
LIN {X 0,Y 114.846,Z 230.179,A -85,B 0,C 180,E1 -25882.701,E2 -25882.701} C_VEL
LIN {X 0,Y 114.863,Z 230.171,A -85,B 0,C 180,E1 -25888.932,E2 -25888.932} C_VEL
LIN {X 0,Y 114.94,Z 230.16,A -85,B 0,C 180,E1 -25896.508,E2 -25896.508} C_VEL
LIN {X 0,Y 115.003,Z 230.159,A -85,B 0,C 180,E1 -25902.21,E2 -25902.21} C_VEL
LIN {X 0,Y 115.249,Z 230.126,A -85,B 0,C 180,E1 -25907.328,E2 -25907.328} C_VEL
LIN {X 0,Y 115.359,Z 230.11,A -85,B 0,C 180,E1 -25913.003,E2 -25913.003} C_VEL
LIN {X 0,Y 115.988,Z 230.034,A -85,B 0,C 180,E1 -25920.002,E2 -25920.002} C_VEL
LIN {X 0,Y 115.384,Z 230.112,A -85,B 0,C 180,E1 -25926.999,E2 -25926.999} C_VEL
LIN {X 0,Y 115.28,Z 230.123,A -85,B 0,C 180,E1 -25932.74,E2 -25932.74} C_VEL
LIN {X 0,Y 115.008,Z 230.154,A -85,B 0,C 180,E1 -25937.793,E2 -25937.793} C_VEL
LIN {X 0,Y 114.944,Z 230.167,A -85,B 0,C 180,E1 -25943.496,E2 -25943.496} C_VEL
LIN {X 0,Y 114.853,Z 230.179,A -85,B 0,C 180,E1 -25951.06,E2 -25951.06} C_VEL
LIN {X 0,Y 114.775,Z 230.188,A -85,B 0,C 180,E1 -25957.76,E2 -25957.76} C_VEL
LIN {X 0,Y 114.889,Z 230.38,A -85,B 0,C 180,E1 -25962.563,E2 -25962.563} C_VEL
LIN {X 0,Y 116.986,Z 239.552,A -85,B 0,C 180,E1 -25968.641,E2 -25968.641} C_VEL
LIN {X 0,Y 119.072,Z 248.902,A -85,B 0,C 180,E1 -25974.397,E2 -25974.397} C_VEL
LIN {X 0,Y 119.647,Z 251.379,A -85,B 0,C 180,E1 -25975.68,E2 -25975.68} C_VEL
LIN {X 0,Y 120.756,Z 256.534,A -85,B 0,C 180,E1 -25976.311,E2 -25976.311} C_VEL
LIN {X 0,Y 120.941,Z 278.392,A -85,B 0,C 180,E1 -25978.293,E2 -25978.293} C_VEL
LIN {X 0,Y 122.166,Z 306.824,A -85,B 0,C 180,E1 -25980.905,E2 -25980.905} C_VEL
LIN {X 0,Y 120.155,Z 350.864,A -85,B 0,C 180,E1 -25984.912,E2 -25984.912} C_VEL
LIN {X 0,Y 119.387,Z 362.734,A -85,B 0,C 180,E1 -25986.59,E2 -25986.59} C_VEL
LIN {X 0,Y 118.176,Z 375.295,A -85,B 0,C 180,E1 -25989.098,E2 -25989.098} C_VEL
LIN {X 0,Y 117.072,Z 386.536,A -85,B 0,C 180,E1 -25992.084,E2 -25992.084} C_VEL
LIN {X 0,Y 116.035,Z 397.772,A -85,B 0,C 180,E1 -25995.982,E2 -25995.982} C_VEL
LIN {X 0,Y 115.531,Z 407.733,A -85,B 0,C 180,E1 -26000.372,E2 -26000.372} C_VEL
LIN {X 0,Y 115.56,Z 415.632,A -85,B 0,C 180,E1 -26004.768,E2 -26004.768} C_VEL
LIN {X 0,Y 115.951,Z 420.882,A -85,B 0,C 180,E1 -26008.266,E2 -26008.266} C_VEL
LIN {X 0,Y 116.265,Z 425.168,A -85,B 0,C 180,E1 -26011.734,E2 -26011.734} C_VEL
LIN {X 0,Y 116.061,Z 426.882,A -85,B 0,C 180,E1 -26013.474,E2 -26013.474} C_VEL
LIN {X 0,Y 114.895,Z 430.927,A -85,B 0,C 180,E1 -26018.799,E2 -26018.799} C_VEL
LIN {X 0,Y 114.818,Z 434.013,A -85,B 0,C 180,E1 -26024.175,E2 -26024.175} C_VEL
LIN {X 0,Y 116.661,Z 436.867,A -85,B 0,C 180,E1 -26031.192,E2 -26031.192} C_VEL
LIN {X 0,Y 120.571,Z 438.403,A -85,B 0,C 180,E1 -26037.798,E2 -26037.798} C_VEL
LIN {X 0,Y 126.273,Z 438.581,A -85,B 0,C 180,E1 -26043.821,E2 -26043.821} C_VEL
LIN {X 0,Y 133.605,Z 437.467,A -85,B 0,C 180,E1 -26049.144,E2 -26049.144} C_VEL
LIN {X 0,Y 142.36,Z 435.017,A -85,B 0,C 180,E1 -26053.723,E2 -26053.723} C_VEL
LIN {X 0,Y 152.281,Z 431.062,A -85,B 0,C 180,E1 -26057.599,E2 -26057.599} C_VEL
LIN {X 0,Y 160.263,Z 427.074,A -85,B 0,C 180,E1 -26060.126,E2 -26060.126} C_VEL
LIN {X 0,Y 168.679,Z 422.043,A -85,B 0,C 180,E1 -26062.341,E2 -26062.341} C_VEL
LIN {X 0,Y 179,Z 414.725,A -85,B 0,C 180,E1 -26064.56,E2 -26064.56} C_VEL
LIN {X 0,Y 188.229,Z 406.853,A -85,B 0,C 180,E1 -26066.179,E2 -26066.179} C_VEL
LIN {X 0,Y 191.729,Z 403.487,A -85,B 0,C 180,E1 -26066.708,E2 -26066.708} C_VEL
LIN {X 0,Y 190.63,Z 404.461,A -85,B 0,C 180,E1 -26066.887,E2 -26066.887} C_VEL
LIN {X 0,Y 184.994,Z 409.326,A -85,B 0,C 180,E1 -26066.789,E2 -26066.789} C_VEL
LIN {X 0,Y 175.99,Z 416.114,A -85,B 0,C 180,E1 -26066.125,E2 -26066.125} C_VEL
LIN {X 0,Y 169.212,Z 420.529,A -85,B 0,C 180,E1 -26065.245,E2 -26065.245} C_VEL
LIN {X 0,Y 167.017,Z 421.844,A -85,B 0,C 180,E1 -26064.827,E2 -26064.827} C_VEL
LIN {X 0,Y 158.666,Z 426.469,A -85,B 0,C 180,E1 -26062.875,E2 -26062.875} C_VEL
LIN {X 0,Y 150.299,Z 430.396,A -85,B 0,C 180,E1 -26060.495,E2 -26060.495} C_VEL
LIN {X 0,Y 142.334,Z 433.405,A -85,B 0,C 180,E1 -26057.789,E2 -26057.789} C_VEL
LIN {X 0,Y 132.592,Z 436.144,A -85,B 0,C 180,E1 -26053.558,E2 -26053.558} C_VEL
LIN {X 0,Y 124.151,Z 437.516,A -85,B 0,C 180,E1 -26048.515,E2 -26048.515} C_VEL
LIN {X 0,Y 117.19,Z 437.58,A -85,B 0,C 180,E1 -26042.668,E2 -26042.668} C_VEL
LIN {X 0,Y 111.99,Z 436.377,A -85,B 0,C 180,E1 -26036.061,E2 -26036.061} C_VEL
LIN {X 0,Y 108.917,Z 433.884,A -85,B 0,C 180,E1 -26028.825,E2 -26028.825} C_VEL
LIN {X 0,Y 108.073,Z 429.972,A -85,B 0,C 180,E1 -26021.253,E2 -26021.253} C_VEL
LIN {X 0,Y 108.863,Z 426.044,A -85,B 0,C 180,E1 -26015.56,E2 -26015.56} C_VEL
LIN {X 0,Y 109.396,Z 424.502,A -85,B 0,C 180,E1 -26013.686,E2 -26013.686} C_VEL
LIN {X 0,Y 109.456,Z 421.558,A -85,B 0,C 180,E1 -26010.922,E2 -26010.922} C_VEL
LIN {X 0,Y 108.9,Z 415.299,A -85,B 0,C 180,E1 -26006.302,E2 -26006.302} C_VEL
LIN {X 0,Y 108.684,Z 407.49,A -85,B 0,C 180,E1 -26001.637,E2 -26001.637} C_VEL
LIN {X 0,Y 108.977,Z 397.951,A -85,B 0,C 180,E1 -25997.049,E2 -25997.049} C_VEL
LIN {X 0,Y 109.943,Z 387.22,A -85,B 0,C 180,E1 -25992.95,E2 -25992.95} C_VEL
LIN {X 0,Y 111.015,Z 375.953,A -85,B 0,C 180,E1 -25989.626,E2 -25989.626} C_VEL
LIN {X 0,Y 112.161,Z 363.922,A -85,B 0,C 180,E1 -25986.947,E2 -25986.947} C_VEL
LIN {X 0,Y 112.952,Z 352.857,A -85,B 0,C 180,E1 -25985.169,E2 -25985.169} C_VEL
LIN {X 0,Y 113.762,Z 333.651,A -85,B 0,C 180,E1 -25983.147,E2 -25983.147} C_VEL
LIN {X 0,Y 115.067,Z 303.608,A -85,B 0,C 180,E1 -25980.315,E2 -25980.315} C_VEL
LIN {X 0,Y 113.647,Z 267.51,A -85,B 0,C 180,E1 -25976.772,E2 -25976.772} C_VEL
LIN {X 0,Y 113.551,Z 256.194,A -85,B 0,C 180,E1 -25975.668,E2 -25975.668} C_VEL
LIN {X 0,Y 112.237,Z 250.69,A -85,B 0,C 180,E1 -25974.888,E2 -25974.888} C_VEL
LIN {X 0,Y 110.04,Z 240.978,A -85,B 0,C 180,E1 -25968.632,E2 -25968.632} C_VEL
LIN {X 0,Y 107.779,Z 231.18,A -85,B 0,C 180,E1 -25961.709,E2 -25961.709} C_VEL
LIN {X 0,Y 107.711,Z 231.067,A -85,B 0,C 180,E1 -25955.963,E2 -25955.963} C_VEL
LIN {X 0,Y 107.789,Z 231.057,A -85,B 0,C 180,E1 -25951.442,E2 -25951.442} C_VEL
LIN {X 0,Y 107.908,Z 231.044,A -85,B 0,C 180,E1 -25943.005,E2 -25943.005} C_VEL
LIN {X 0,Y 108.032,Z 231.028,A -85,B 0,C 180,E1 -25935.085,E2 -25935.085} C_VEL
LIN {X 0,Y 108.283,Z 230.99,A -85,B 0,C 180,E1 -25931.23,E2 -25931.23} C_VEL
LIN {X 0,Y 108.452,Z 230.972,A -85,B 0,C 180,E1 -25923.717,E2 -25923.717} C_VEL
LIN {X 0,Y 108.937,Z 230.912,A -85,B 0,C 180,E1 -25920.002,E2 -25920.002} C_VEL
LIN {X 0,Y 108.298,Z 230.99,A -85,B 0,C 180,E1 -25912.544,E2 -25912.544} C_VEL
LIN {X 0,Y 108.169,Z 231.008,A -85,B 0,C 180,E1 -25907.041,E2 -25907.041} C_VEL
LIN {X 0,Y 107.896,Z 231.045,A -85,B 0,C 180,E1 -25900.995,E2 -25900.995} C_VEL
LIN {X 0,Y 107.851,Z 231.045,A -85,B 0,C 180,E1 -25895.816,E2 -25895.816} C_VEL
LIN {X 0,Y 107.793,Z 231.052,A -85,B 0,C 180,E1 -25887.944,E2 -25887.944} C_VEL
LIN {X 0,Y 107.745,Z 231.059,A -85,B 0,C 180,E1 -25881.507,E2 -25881.507} C_VEL
LIN {X 0,Y 107.762,Z 231.06,A -85,B 0,C 180,E1 -25874.163,E2 -25874.163} C_VEL
LIN {X 0,Y 107.75,Z 231.063,A -85,B 0,C 180,E1 -25868.494,E2 -25868.494} C_VEL
LIN {X 0,Y 107.806,Z 231.053,A -85,B 0,C 180,E1 -25861.432,E2 -25861.432} C_VEL
LIN {X 0,Y 107.906,Z 231.04,A -85,B 0,C 180,E1 -25853,E2 -25853} C_VEL
LIN {X 0,Y 108.033,Z 231.023,A -85,B 0,C 180,E1 -25845.08,E2 -25845.08} C_VEL
LIN {X 0,Y 108.285,Z 230.997,A -85,B 0,C 180,E1 -25841.225,E2 -25841.225} C_VEL
LIN {X 0,Y 108.455,Z 230.975,A -85,B 0,C 180,E1 -25833.713,E2 -25833.713} C_VEL
LIN {X 0,Y 108.943,Z 230.908,A -85,B 0,C 180,E1 -25829.997,E2 -25829.997} C_VEL
LIN {X 0,Y 108.337,Z 230.985,A -85,B 0,C 180,E1 -25822.543,E2 -25822.543} C_VEL
LIN {X 0,Y 108.201,Z 231.007,A -85,B 0,C 180,E1 -25816.972,E2 -25816.972} C_VEL
LIN {X 0,Y 107.905,Z 231.045,A -85,B 0,C 180,E1 -25810.992,E2 -25810.992} C_VEL
LIN {X 0,Y 107.859,Z 231.05,A -85,B 0,C 180,E1 -25805.811,E2 -25805.811} C_VEL
LIN {X 0,Y 107.946,Z 231.206,A -85,B 0,C 180,E1 -25798.881,E2 -25798.881} C_VEL
LIN {X 0,Y 109.48,Z 238.177,A -85,B 0,C 180,E1 -25793.57,E2 -25793.57} C_VEL
LIN {X 0,Y 110.079,Z 241.202,A -85,B 0,C 180,E1 -25791.645,E2 -25791.645} C_VEL
LIN {X 0,Y 114,Z 257.22,A -85,B 0,C 180,E1 -25789.585,E2 -25789.585} C_VEL
LIN {X 0,Y 115.259,Z 271.38,A -85,B 0,C 180,E1 -25788.058,E2 -25788.058} C_VEL
LIN {X 0,Y 111.77,Z 333.529,A -85,B 0,C 180,E1 -25781.763,E2 -25781.763} C_VEL
LIN {X 0,Y 110.797,Z 346.008,A -85,B 0,C 180,E1 -25779.807,E2 -25779.807} C_VEL
LIN {X 0,Y 109.776,Z 356.936,A -85,B 0,C 180,E1 -25777.457,E2 -25777.457} C_VEL
LIN {X 0,Y 108.561,Z 368.999,A -85,B 0,C 180,E1 -25774.072,E2 -25774.072} C_VEL
LIN {X 0,Y 107.493,Z 380.44,A -85,B 0,C 180,E1 -25769.901,E2 -25769.901} C_VEL
LIN {X 0,Y 106.83,Z 390.375,A -85,B 0,C 180,E1 -25765.314,E2 -25765.314} C_VEL
LIN {X 0,Y 106.466,Z 399.407,A -85,B 0,C 180,E1 -25760.092,E2 -25760.092} C_VEL
LIN {X 0,Y 107.044,Z 407.584,A -85,B 0,C 180,E1 -25754.154,E2 -25754.154} C_VEL
LIN {X 0,Y 108.411,Z 413.138,A -85,B 0,C 180,E1 -25749.325,E2 -25749.325} C_VEL
LIN {X 0,Y 111.084,Z 418.617,A -85,B 0,C 180,E1 -25743.626,E2 -25743.626} C_VEL
LIN {X 0,Y 114.887,Z 422.756,A -85,B 0,C 180,E1 -25738.246,E2 -25738.246} C_VEL
LIN {X 0,Y 120.475,Z 426.105,A -85,B 0,C 180,E1 -25732.63,E2 -25732.63} C_VEL
LIN {X 0,Y 123.555,Z 427.203,A -85,B 0,C 180,E1 -25730.173,E2 -25730.173} C_VEL
LIN {X 0,Y 130.661,Z 428.451,A -85,B 0,C 180,E1 -25725.514,E2 -25725.514} C_VEL
LIN {X 0,Y 137.211,Z 428.518,A -85,B 0,C 180,E1 -25722.101,E2 -25722.101} C_VEL
LIN {X 0,Y 142.349,Z 427.999,A -85,B 0,C 180,E1 -25719.78,E2 -25719.78} C_VEL
LIN {X 0,Y 147.797,Z 427.019,A -85,B 0,C 180,E1 -25717.639,E2 -25717.639} C_VEL
LIN {X 0,Y 154.785,Z 425.1,A -85,B 0,C 180,E1 -25715.247,E2 -25715.247} C_VEL
LIN {X 0,Y 162.503,Z 422.168,A -85,B 0,C 180,E1 -25712.991,E2 -25712.991} C_VEL
LIN {X 0,Y 171.97,Z 417.53,A -85,B 0,C 180,E1 -25710.631,E2 -25710.631} C_VEL
LIN {X 0,Y 181.021,Z 411.867,A -85,B 0,C 180,E1 -25708.666,E2 -25708.666} C_VEL
LIN {X 0,Y 182.833,Z 410.722,A -85,B 0,C 180,E1 -25707.746,E2 -25707.746} C_VEL
LIN {X 0,Y 173.505,Z 417.695,A -85,B 0,C 180,E1 -25706.139,E2 -25706.139} C_VEL
LIN {X 0,Y 167.017,Z 421.844,A -85,B 0,C 180,E1 -25704.827,E2 -25704.827} C_VEL
LIN {X 0,Y 162.2,Z 424.514,A -85,B 0,C 180,E1 -25704.028,E2 -25704.028} C_VEL
LIN {X 0,Y 149.836,Z 429.691,A -85,B 0,C 180,E1 -25702.69,E2 -25702.69} C_VEL
LIN {X 0,Y 142.899,Z 431.938,A -85,B 0,C 180,E1 -25701.554,E2 -25701.554} C_VEL
LIN {X 0,Y 139.769,Z 432.826,A -85,B 0,C 180,E1 -25700.691,E2 -25700.691} C_VEL
LIN {X 0,Y 132.47,Z 434.774,A -85,B 0,C 180,E1 -25697.968,E2 -25697.968} C_VEL
LIN {X 0,Y 122.957,Z 436.39,A -85,B 0,C 180,E1 -25693.309,E2 -25693.309} C_VEL
LIN {X 0,Y 114.813,Z 436.723,A -85,B 0,C 180,E1 -25687.746,E2 -25687.746} C_VEL
LIN {X 0,Y 108.329,Z 435.787,A -85,B 0,C 180,E1 -25681.269,E2 -25681.269} C_VEL
LIN {X 0,Y 103.817,Z 433.576,A -85,B 0,C 180,E1 -25673.968,E2 -25673.968} C_VEL
LIN {X 0,Y 101.569,Z 430.078,A -85,B 0,C 180,E1 -25666.071,E2 -25666.071} C_VEL
LIN {X 0,Y 101.847,Z 425.056,A -85,B 0,C 180,E1 -25657.935,E2 -25657.935} C_VEL
LIN {X 0,Y 102.773,Z 421.941,A -85,B 0,C 180,E1 -25653.924,E2 -25653.924} C_VEL
LIN {X 0,Y 102.696,Z 418.802,A -85,B 0,C 180,E1 -25650.983,E2 -25650.983} C_VEL
LIN {X 0,Y 102.035,Z 412.058,A -85,B 0,C 180,E1 -25646.053,E2 -25646.053} C_VEL
LIN {X 0,Y 101.907,Z 403.667,A -85,B 0,C 180,E1 -25641.076,E2 -25641.076} C_VEL
LIN {X 0,Y 102.278,Z 394.431,A -85,B 0,C 180,E1 -25636.637,E2 -25636.637} C_VEL
LIN {X 0,Y 103.154,Z 383.881,A -85,B 0,C 180,E1 -25632.611,E2 -25632.611} C_VEL
LIN {X 0,Y 104.225,Z 372.653,A -85,B 0,C 180,E1 -25629.27,E2 -25629.27} C_VEL
LIN {X 0,Y 105.454,Z 359.7,A -85,B 0,C 180,E1 -25626.433,E2 -25626.433} C_VEL
LIN {X 0,Y 106.168,Z 347.056,A -85,B 0,C 180,E1 -25624.518,E2 -25624.518} C_VEL
LIN {X 0,Y 107.997,Z 303.774,A -85,B 0,C 180,E1 -25620.036,E2 -25620.036} C_VEL
LIN {X 0,Y 106.624,Z 267.833,A -85,B 0,C 180,E1 -25616.275,E2 -25616.275} C_VEL
LIN {X 0,Y 106.671,Z 257.743,A -85,B 0,C 180,E1 -25615.238,E2 -25615.238} C_VEL
LIN {X 0,Y 104.919,Z 250.498,A -85,B 0,C 180,E1 -25614.211,E2 -25614.211} C_VEL
LIN {X 0,Y 103.053,Z 242.288,A -85,B 0,C 180,E1 -25608.608,E2 -25608.608} C_VEL
LIN {X 0,Y 100.912,Z 232.98,A -85,B 0,C 180,E1 -25601.71,E2 -25601.71} C_VEL
LIN {X 0,Y 100.7,Z 231.995,A -85,B 0,C 180,E1 -25600.631,E2 -25600.631} C_VEL
LIN {X 0,Y 100.686,Z 231.941,A -85,B 0,C 180,E1 -25593.117,E2 -25593.117} C_VEL
LIN {X 0,Y 100.783,Z 231.93,A -85,B 0,C 180,E1 -25584.736,E2 -25584.736} C_VEL
LIN {X 0,Y 100.813,Z 231.924,A -85,B 0,C 180,E1 -25580.402,E2 -25580.402} C_VEL
LIN {X 0,Y 101.183,Z 231.877,A -85,B 0,C 180,E1 -25572.029,E2 -25572.029} C_VEL
LIN {X 0,Y 101.262,Z 231.869,A -85,B 0,C 180,E1 -25567.981,E2 -25567.981} C_VEL
LIN {X 0,Y 101.861,Z 231.794,A -85,B 0,C 180,E1 -25560.002,E2 -25560.002} C_VEL
LIN {X 0,Y 101.237,Z 231.87,A -85,B 0,C 180,E1 -25552.021,E2 -25552.021} C_VEL
LIN {X 0,Y 101.098,Z 231.888,A -85,B 0,C 180,E1 -25546.699,E2 -25546.699} C_VEL
LIN {X 0,Y 100.808,Z 231.926,A -85,B 0,C 180,E1 -25539.601,E2 -25539.601} C_VEL
LIN {X 0,Y 100.768,Z 231.93,A -85,B 0,C 180,E1 -25535.042,E2 -25535.042} C_VEL
LIN {X 0,Y 100.701,Z 231.937,A -85,B 0,C 180,E1 -25526.87,E2 -25526.87} C_VEL
LIN {X 0,Y 100.692,Z 231.935,A -85,B 0,C 180,E1 -25520.148,E2 -25520.148} C_VEL
LIN {X 0,Y 100.728,Z 231.936,A -85,B 0,C 180,E1 -25514.24,E2 -25514.24} C_VEL
LIN {X 0,Y 100.69,Z 231.941,A -85,B 0,C 180,E1 -25508.912,E2 -25508.912} C_VEL
LIN {X 0,Y 100.702,Z 231.933,A -85,B 0,C 180,E1 -25503.129,E2 -25503.129} C_VEL
LIN {X 0,Y 100.781,Z 231.924,A -85,B 0,C 180,E1 -25494.731,E2 -25494.731} C_VEL
LIN {X 0,Y 100.812,Z 231.927,A -85,B 0,C 180,E1 -25490.397,E2 -25490.397} C_VEL
LIN {X 0,Y 101.184,Z 231.881,A -85,B 0,C 180,E1 -25482.024,E2 -25482.024} C_VEL
LIN {X 0,Y 101.264,Z 231.863,A -85,B 0,C 180,E1 -25477.976,E2 -25477.976} C_VEL
LIN {X 0,Y 101.868,Z 231.789,A -85,B 0,C 180,E1 -25469.997,E2 -25469.997} C_VEL
LIN {X 0,Y 101.277,Z 231.864,A -85,B 0,C 180,E1 -25462.02,E2 -25462.02} C_VEL
LIN {X 0,Y 101.127,Z 231.888,A -85,B 0,C 180,E1 -25456.635,E2 -25456.635} C_VEL
LIN {X 0,Y 100.816,Z 231.928,A -85,B 0,C 180,E1 -25449.598,E2 -25449.598} C_VEL
LIN {X 0,Y 100.774,Z 231.931,A -85,B 0,C 180,E1 -25445.038,E2 -25445.038} C_VEL
LIN {X 0,Y 100.911,Z 232.078,A -85,B 0,C 180,E1 -25439.67,E2 -25439.67} C_VEL
LIN {X 0,Y 102.274,Z 238.393,A -85,B 0,C 180,E1 -25434.5,E2 -25434.5} C_VEL
LIN {X 0,Y 102.887,Z 241.382,A -85,B 0,C 180,E1 -25432.402,E2 -25432.402} C_VEL
LIN {X 0,Y 107.043,Z 258.354,A -85,B 0,C 180,E1 -25430.041,E2 -25430.041} C_VEL
LIN {X 0,Y 108.228,Z 271.605,A -85,B 0,C 180,E1 -25428.531,E2 -25428.531} C_VEL
LIN {X 0,Y 104.609,Z 334.003,A -85,B 0,C 180,E1 -25421.721,E2 -25421.721} C_VEL
LIN {X 0,Y 103.596,Z 347.197,A -85,B 0,C 180,E1 -25419.492,E2 -25419.492} C_VEL
LIN {X 0,Y 102.323,Z 360.411,A -85,B 0,C 180,E1 -25416.323,E2 -25416.323} C_VEL
LIN {X 0,Y 101.158,Z 372.095,A -85,B 0,C 180,E1 -25412.575,E2 -25412.575} C_VEL
LIN {X 0,Y 100.252,Z 382.682,A -85,B 0,C 180,E1 -25408.24,E2 -25408.24} C_VEL
LIN {X 0,Y 99.742,Z 391.602,A -85,B 0,C 180,E1 -25403.646,E2 -25403.646} C_VEL
LIN {X 0,Y 99.572,Z 399.771,A -85,B 0,C 180,E1 -25398.517,E2 -25398.517} C_VEL
